LIN {X 0,Y 468.722,Z 59.104,A -85,B 0,C 180,E1 -7454.434,E2 -7454.434} C_VEL
LIN {X 0,Y 467.684,Z 59.23,A -85,B 0,C 180,E1 -7455.151,E2 -7455.151} C_VEL
LIN {X 0,Y 467.596,Z 59.24,A -85,B 0,C 180,E1 -7455.394,E2 -7455.394} C_VEL
LIN {X 0,Y 467.647,Z 59.28,A -85,B 0,C 180,E1 -7456.807,E2 -7456.807} C_VEL
LIN {X 0,Y 468.564,Z 66.05,A -85,B 0,C 180,E1 -7458.318,E2 -7458.318} C_VEL
LIN {X 0,Y 468.563,Z 74.796,A -85,B 0,C 180,E1 -7460.187,E2 -7460.187} C_VEL
LIN {X 0,Y 471.18,Z 89.776,A -85,B 0,C 180,E1 -7460.508,E2 -7460.508} C_VEL
LIN {X 0,Y 470.424,Z 181.464,A -85,B 0,C 180,E1 -7461.922,E2 -7461.922} C_VEL
LIN {X 0,Y 470.218,Z 194.57,A -85,B 0,C 180,E1 -7462.297,E2 -7462.297} C_VEL
LIN {X 0,Y 469.826,Z 207.741,A -85,B 0,C 180,E1 -7462.857,E2 -7462.857} C_VEL
LIN {X 0,Y 469.579,Z 219.557,A -85,B 0,C 180,E1 -7463.555,E2 -7463.555} C_VEL
LIN {X 0,Y 469.031,Z 230.914,A -85,B 0,C 180,E1 -7464.411,E2 -7464.411} C_VEL
LIN {X 0,Y 468.581,Z 241.141,A -85,B 0,C 180,E1 -7465.376,E2 -7465.376} C_VEL
LIN {X 0,Y 468.212,Z 249.513,A -85,B 0,C 180,E1 -7466.343,E2 -7466.343} C_VEL
LIN {X 0,Y 467.732,Z 258.606,A -85,B 0,C 180,E1 -7467.632,E2 -7467.632} C_VEL
LIN {X 0,Y 467.395,Z 265.922,A -85,B 0,C 180,E1 -7468.923,E2 -7468.923} C_VEL
LIN {X 0,Y 467.046,Z 272.679,A -85,B 0,C 180,E1 -7470.431,E2 -7470.431} C_VEL
LIN {X 0,Y 466.837,Z 277.14,A -85,B 0,C 180,E1 -7471.726,E2 -7471.726} C_VEL
LIN {X 0,Y 466.857,Z 279.486,A -85,B 0,C 180,E1 -7472.589,E2 -7472.589} C_VEL
LIN {X 0,Y 466.812,Z 281.417,A -85,B 0,C 180,E1 -7473.453,E2 -7473.453} C_VEL
LIN {X 0,Y 466.694,Z 282.945,A -85,B 0,C 180,E1 -7474.318,E2 -7474.318} C_VEL
LIN {X 0,Y 466.717,Z 284.018,A -85,B 0,C 180,E1 -7475.184,E2 -7475.184} C_VEL
LIN {X 0,Y 466.747,Z 284.88,A -85,B 0,C 180,E1 -7476.385,E2 -7476.385} C_VEL
LIN {X 0,Y 466.689,Z 284.914,A -85,B 0,C 180,E1 -7477.79,E2 -7477.79} C_VEL
LIN {X 0,Y 466.685,Z 284.397,A -85,B 0,C 180,E1 -7478.662,E2 -7478.662} C_VEL
LIN {X 0,Y 466.724,Z 282.165,A -85,B 0,C 180,E1 -7480.411,E2 -7480.411} C_VEL
LIN {X 0,Y 466.916,Z 278.848,A -85,B 0,C 180,E1 -7481.934,E2 -7481.934} C_VEL
LIN {X 0,Y 467.093,Z 273.978,A -85,B 0,C 180,E1 -7483.487,E2 -7483.487} C_VEL
LIN {X 0,Y 467.477,Z 267.522,A -85,B 0,C 180,E1 -7485.031,E2 -7485.031} C_VEL
LIN {X 0,Y 467.808,Z 260.476,A -85,B 0,C 180,E1 -7486.349,E2 -7486.349} C_VEL
LIN {X 0,Y 468.253,Z 251.445,A -85,B 0,C 180,E1 -7487.694,E2 -7487.694} C_VEL
LIN {X 0,Y 468.777,Z 242.455,A -85,B 0,C 180,E1 -7488.777,E2 -7488.777} C_VEL
LIN {X 0,Y 469.253,Z 231.889,A -85,B 0,C 180,E1 -7489.807,E2 -7489.807} C_VEL
LIN {X 0,Y 469.773,Z 220.35,A -85,B 0,C 180,E1 -7490.698,E2 -7490.698} C_VEL
LIN {X 0,Y 470.294,Z 208.288,A -85,B 0,C 180,E1 -7491.42,E2 -7491.42} C_VEL
LIN {X 0,Y 470.684,Z 195.785,A -85,B 0,C 180,E1 -7491.967,E2 -7491.967} C_VEL
LIN {X 0,Y 470.974,Z 182.953,A -85,B 0,C 180,E1 -7492.349,E2 -7492.349} C_VEL
LIN {X 0,Y 471.195,Z 149.03,A -85,B 0,C 180,E1 -7492.905,E2 -7492.905} C_VEL
LIN {X 0,Y 471.683,Z 88.302,A -85,B 0,C 180,E1 -7493.841,E2 -7493.841} C_VEL
LIN {X 0,Y 468.749,Z 74.914,A -85,B 0,C 180,E1 -7494.191,E2 -7494.191} C_VEL
LIN {X 0,Y 468.9,Z 66.893,A -85,B 0,C 180,E1 -7495.933,E2 -7495.933} C_VEL
LIN {X 0,Y 467.611,Z 59.24,A -85,B 0,C 180,E1 -7497.729,E2 -7497.729} C_VEL
LIN {X 0,Y 467.544,Z 59.245,A -85,B 0,C 180,E1 -7501.039,E2 -7501.039} C_VEL
LIN {X 0,Y 467.566,Z 59.245,A -85,B 0,C 180,E1 -7504.237,E2 -7504.237} C_VEL
LIN {X 0,Y 467.516,Z 59.246,A -85,B 0,C 180,E1 -7507.18,E2 -7507.18} C_VEL
LIN {X 0,Y 467.541,Z 59.247,A -85,B 0,C 180,E1 -7510.269,E2 -7510.269} C_VEL
LIN {X 0,Y 467.519,Z 59.247,A -85,B 0,C 180,E1 -7512.568,E2 -7512.568} C_VEL
LIN {X 0,Y 467.565,Z 59.232,A -85,B 0,C 180,E1 -7515.052,E2 -7515.052} C_VEL
LIN {X 0,Y 467.553,Z 59.239,A -85,B 0,C 180,E1 -7518.727,E2 -7518.727} C_VEL
LIN {X 0,Y 467.534,Z 59.246,A -85,B 0,C 180,E1 -7521.952,E2 -7521.952} C_VEL
LIN {X 0,Y 467.543,Z 59.244,A -85,B 0,C 180,E1 -7525.165,E2 -7525.165} C_VEL
LIN {X 0,Y 467.545,Z 59.239,A -85,B 0,C 180,E1 -7528.257,E2 -7528.257} C_VEL
LIN {X 0,Y 467.53,Z 59.248,A -85,B 0,C 180,E1 -7531.247,E2 -7531.247} C_VEL
LIN {X 0,Y 467.564,Z 59.24,A -85,B 0,C 180,E1 -7534.405,E2 -7534.405} C_VEL
LIN {X 0,Y 467.575,Z 59.24,A -85,B 0,C 180,E1 -7536.995,E2 -7536.995} C_VEL
LIN {X 0,Y 467.623,Z 59.232,A -85,B 0,C 180,E1 -7539.777,E2 -7539.777} C_VEL
LIN {X 0,Y 467.594,Z 59.236,A -85,B 0,C 180,E1 -7542.506,E2 -7542.506} C_VEL
LIN {X 0,Y 467.598,Z 59.237,A -85,B 0,C 180,E1 -7545.196,E2 -7545.196} C_VEL
LIN {X 0,Y 467.659,Z 59.223,A -85,B 0,C 180,E1 -7547.854,E2 -7547.854} C_VEL
LIN {X 0,Y 467.66,Z 59.228,A -85,B 0,C 180,E1 -7551.357,E2 -7551.357} C_VEL
LIN {X 0,Y 467.696,Z 59.22,A -85,B 0,C 180,E1 -7553.962,E2 -7553.962} C_VEL
LIN {X 0,Y 467.826,Z 59.207,A -85,B 0,C 180,E1 -7557.417,E2 -7557.417} C_VEL
LIN {X 0,Y 467.852,Z 59.203,A -85,B 0,C 180,E1 -7560,E2 -7560} C_VEL
LIN {X 0,Y 467.816,Z 59.21,A -85,B 0,C 180,E1 -7562.583,E2 -7562.583} C_VEL
LIN {X 0,Y 467.706,Z 59.221,A -85,B 0,C 180,E1 -7566.038,E2 -7566.038} C_VEL
LIN {X 0,Y 467.661,Z 59.227,A -85,B 0,C 180,E1 -7568.643,E2 -7568.643} C_VEL
LIN {X 0,Y 467.66,Z 59.227,A -85,B 0,C 180,E1 -7572.145,E2 -7572.145} C_VEL
LIN {X 0,Y 467.64,Z 59.233,A -85,B 0,C 180,E1 -7575.695,E2 -7575.695} C_VEL
LIN {X 0,Y 467.623,Z 59.236,A -85,B 0,C 180,E1 -7579.308,E2 -7579.308} C_VEL
LIN {X 0,Y 467.537,Z 59.239,A -85,B 0,C 180,E1 -7582.074,E2 -7582.074} C_VEL
LIN {X 0,Y 467.572,Z 59.242,A -85,B 0,C 180,E1 -7584.889,E2 -7584.889} C_VEL
LIN {X 0,Y 467.618,Z 59.234,A -85,B 0,C 180,E1 -7587.769,E2 -7587.769} C_VEL
LIN {X 0,Y 467.57,Z 59.242,A -85,B 0,C 180,E1 -7591.044,E2 -7591.044} C_VEL
LIN {X 0,Y 467.591,Z 59.236,A -85,B 0,C 180,E1 -7594.242,E2 -7594.242} C_VEL
LIN {X 0,Y 467.55,Z 59.238,A -85,B 0,C 180,E1 -7597.186,E2 -7597.186} C_VEL
LIN {X 0,Y 467.577,Z 59.241,A -85,B 0,C 180,E1 -7600.265,E2 -7600.265} C_VEL
LIN {X 0,Y 467.589,Z 59.243,A -85,B 0,C 180,E1 -7602.567,E2 -7602.567} C_VEL
LIN {X 0,Y 467.568,Z 59.241,A -85,B 0,C 180,E1 -7605.052,E2 -7605.052} C_VEL
LIN {X 0,Y 467.592,Z 59.235,A -85,B 0,C 180,E1 -7607.44,E2 -7607.44} C_VEL
LIN {X 0,Y 467.585,Z 59.239,A -85,B 0,C 180,E1 -7610.855,E2 -7610.855} C_VEL
LIN {X 0,Y 467.562,Z 59.242,A -85,B 0,C 180,E1 -7614.261,E2 -7614.261} C_VEL
LIN {X 0,Y 467.585,Z 59.242,A -85,B 0,C 180,E1 -7617.321,E2 -7617.321} C_VEL
LIN {X 0,Y 467.572,Z 59.244,A -85,B 0,C 180,E1 -7620.667,E2 -7620.667} C_VEL
LIN {X 0,Y 467.696,Z 59.391,A -85,B 0,C 180,E1 -7623.295,E2 -7623.295} C_VEL
LIN {X 0,Y 470.046,Z 71.407,A -85,B 0,C 180,E1 -7625.579,E2 -7625.579} C_VEL
LIN {X 0,Y 469.737,Z 81.506,A -85,B 0,C 180,E1 -7627.34,E2 -7627.34} C_VEL
LIN {X 0,Y 468.798,Z 101.855,A -85,B 0,C 180,E1 -7630.816,E2 -7630.816} C_VEL
LIN {X 0,Y 468.334,Z 113.848,A -85,B 0,C 180,E1 -7632.842,E2 -7632.842} C_VEL
LIN {X 0,Y 471.406,Z 134.719,A -85,B 0,C 180,E1 -7633.296,E2 -7633.296} C_VEL
LIN {X 0,Y 470.758,Z 222.171,A -85,B 0,C 180,E1 -7634.661,E2 -7634.661} C_VEL
LIN {X 0,Y 470.321,Z 235.512,A -85,B 0,C 180,E1 -7635.034,E2 -7635.034} C_VEL
LIN {X 0,Y 469.848,Z 247.706,A -85,B 0,C 180,E1 -7635.545,E2 -7635.545} C_VEL
LIN {X 0,Y 469.32,Z 260.024,A -85,B 0,C 180,E1 -7636.247,E2 -7636.247} C_VEL
LIN {X 0,Y 468.688,Z 271.899,A -85,B 0,C 180,E1 -7637.133,E2 -7637.133} C_VEL
LIN {X 0,Y 468.246,Z 282.11,A -85,B 0,C 180,E1 -7638.09,E2 -7638.09} C_VEL
LIN {X 0,Y 467.715,Z 291.557,A -85,B 0,C 180,E1 -7639.174,E2 -7639.174} C_VEL
LIN {X 0,Y 467.305,Z 300.678,A -85,B 0,C 180,E1 -7640.477,E2 -7640.477} C_VEL
LIN {X 0,Y 466.988,Z 308.043,A -85,B 0,C 180,E1 -7641.78,E2 -7641.78} C_VEL
LIN {X 0,Y 466.824,Z 313.963,A -85,B 0,C 180,E1 -7643.082,E2 -7643.082} C_VEL
LIN {X 0,Y 466.709,Z 318.64,A -85,B 0,C 180,E1 -7644.383,E2 -7644.383} C_VEL
LIN {X 0,Y 466.646,Z 322.21,A -85,B 0,C 180,E1 -7645.681,E2 -7645.681} C_VEL
LIN {X 0,Y 466.699,Z 324.041,A -85,B 0,C 180,E1 -7646.546,E2 -7646.546} C_VEL
LIN {X 0,Y 466.684,Z 325.418,A -85,B 0,C 180,E1 -7647.41,E2 -7647.41} C_VEL
LIN {X 0,Y 466.664,Z 326.4,A -85,B 0,C 180,E1 -7648.274,E2 -7648.274} C_VEL
LIN {X 0,Y 466.63,Z 326.992,A -85,B 0,C 180,E1 -7649.137,E2 -7649.137} C_VEL
LIN {X 0,Y 466.614,Z 327.175,A -85,B 0,C 180,E1 -7650,E2 -7650} C_VEL
LIN {X 0,Y 466.664,Z 326.308,A -85,B 0,C 180,E1 -7651.726,E2 -7651.726} C_VEL
LIN {X 0,Y 466.685,Z 325.29,A -85,B 0,C 180,E1 -7652.589,E2 -7652.589} C_VEL
LIN {X 0,Y 466.73,Z 323.852,A -85,B 0,C 180,E1 -7653.453,E2 -7653.453} C_VEL
LIN {X 0,Y 466.685,Z 320.859,A -85,B 0,C 180,E1 -7654.751,E2 -7654.751} C_VEL
LIN {X 0,Y 466.704,Z 315.725,A -85,B 0,C 180,E1 -7656.341,E2 -7656.341} C_VEL
LIN {X 0,Y 466.927,Z 309.562,A -85,B 0,C 180,E1 -7657.785,E2 -7657.785} C_VEL
LIN {X 0,Y 467.158,Z 302.53,A -85,B 0,C 180,E1 -7659.088,E2 -7659.088} C_VEL
LIN {X 0,Y 467.465,Z 293.71,A -85,B 0,C 180,E1 -7660.393,E2 -7660.393} C_VEL
LIN {X 0,Y 468.005,Z 283.701,A -85,B 0,C 180,E1 -7661.587,E2 -7661.587} C_VEL
LIN {X 0,Y 468.432,Z 273.768,A -85,B 0,C 180,E1 -7662.542,E2 -7662.542} C_VEL
LIN {X 0,Y 468.936,Z 262.165,A -85,B 0,C 180,E1 -7663.432,E2 -7663.432} C_VEL
LIN {X 0,Y 469.429,Z 250.422,A -85,B 0,C 180,E1 -7664.136,E2 -7664.136} C_VEL
LIN {X 0,Y 469.88,Z 237.655,A -85,B 0,C 180,E1 -7664.702,E2 -7664.702} C_VEL
LIN {X 0,Y 470.294,Z 224.05,A -85,B 0,C 180,E1 -7665.104,E2 -7665.104} C_VEL
LIN {X 0,Y 470.602,Z 188.382,A -85,B 0,C 180,E1 -7665.677,E2 -7665.677} C_VEL
LIN {X 0,Y 470.79,Z 132.877,A -85,B 0,C 180,E1 -7666.528,E2 -7666.528} C_VEL
LIN {X 0,Y 468.138,Z 113.96,A -85,B 0,C 180,E1 -7666.918,E2 -7666.918} C_VEL
LIN {X 0,Y 468.755,Z 95.783,A -85,B 0,C 180,E1 -7669.943,E2 -7669.943} C_VEL
LIN {X 0,Y 469.614,Z 75.42,A -85,B 0,C 180,E1 -7673.365,E2 -7673.365} C_VEL
LIN {X 0,Y 469.599,Z 69.43,A -85,B 0,C 180,E1 -7674.394,E2 -7674.394} C_VEL
LIN {X 0,Y 467.643,Z 59.237,A -85,B 0,C 180,E1 -7676.257,E2 -7676.257} C_VEL
LIN {X 0,Y 467.571,Z 59.242,A -85,B 0,C 180,E1 -7679.332,E2 -7679.332} C_VEL
LIN {X 0,Y 467.582,Z 59.237,A -85,B 0,C 180,E1 -7682.679,E2 -7682.679} C_VEL
LIN {X 0,Y 467.56,Z 59.247,A -85,B 0,C 180,E1 -7685.739,E2 -7685.739} C_VEL
LIN {X 0,Y 467.583,Z 59.238,A -85,B 0,C 180,E1 -7689.144,E2 -7689.144} C_VEL
LIN {X 0,Y 467.586,Z 59.236,A -85,B 0,C 180,E1 -7692.567,E2 -7692.567} C_VEL
LIN {X 0,Y 467.565,Z 59.241,A -85,B 0,C 180,E1 -7695.052,E2 -7695.052} C_VEL
LIN {X 0,Y 467.588,Z 59.244,A -85,B 0,C 180,E1 -7697.44,E2 -7697.44} C_VEL
LIN {X 0,Y 467.575,Z 59.24,A -85,B 0,C 180,E1 -7700.855,E2 -7700.855} C_VEL
LIN {X 0,Y 467.56,Z 59.239,A -85,B 0,C 180,E1 -7704.261,E2 -7704.261} C_VEL
LIN {X 0,Y 467.581,Z 59.242,A -85,B 0,C 180,E1 -7707.321,E2 -7707.321} C_VEL
LIN {X 0,Y 467.569,Z 59.242,A -85,B 0,C 180,E1 -7710.667,E2 -7710.667} C_VEL
LIN {X 0,Y 467.616,Z 59.237,A -85,B 0,C 180,E1 -7713.2,E2 -7713.2} C_VEL
LIN {X 0,Y 467.591,Z 59.239,A -85,B 0,C 180,E1 -7716.468,E2 -7716.468} C_VEL
LIN {X 0,Y 467.622,Z 59.232,A -85,B 0,C 180,E1 -7719.777,E2 -7719.777} C_VEL
LIN {X 0,Y 467.597,Z 59.241,A -85,B 0,C 180,E1 -7722.506,E2 -7722.506} C_VEL
LIN {X 0,Y 467.604,Z 59.235,A -85,B 0,C 180,E1 -7725.196,E2 -7725.196} C_VEL
LIN {X 0,Y 467.656,Z 59.229,A -85,B 0,C 180,E1 -7727.855,E2 -7727.855} C_VEL
LIN {X 0,Y 467.679,Z 59.224,A -85,B 0,C 180,E1 -7731.357,E2 -7731.357} C_VEL
LIN {X 0,Y 467.736,Z 59.221,A -85,B 0,C 180,E1 -7733.963,E2 -7733.963} C_VEL
LIN {X 0,Y 467.852,Z 59.203,A -85,B 0,C 180,E1 -7737.417,E2 -7737.417} C_VEL
LIN {X 0,Y 467.881,Z 59.206,A -85,B 0,C 180,E1 -7740,E2 -7740} C_VEL
LIN {X 0,Y 467.852,Z 59.204,A -85,B 0,C 180,E1 -7742.583,E2 -7742.583} C_VEL
LIN {X 0,Y 467.721,Z 59.225,A -85,B 0,C 180,E1 -7746.038,E2 -7746.038} C_VEL
LIN {X 0,Y 467.669,Z 59.226,A -85,B 0,C 180,E1 -7748.643,E2 -7748.643} C_VEL
LIN {X 0,Y 467.656,Z 59.23,A -85,B 0,C 180,E1 -7752.146,E2 -7752.146} C_VEL
LIN {X 0,Y 467.639,Z 59.236,A -85,B 0,C 180,E1 -7755.695,E2 -7755.695} C_VEL
LIN {X 0,Y 467.621,Z 59.237,A -85,B 0,C 180,E1 -7759.308,E2 -7759.308} C_VEL
LIN {X 0,Y 467.534,Z 59.243,A -85,B 0,C 180,E1 -7762.074,E2 -7762.074} C_VEL
LIN {X 0,Y 467.569,Z 59.241,A -85,B 0,C 180,E1 -7764.89,E2 -7764.89} C_VEL
LIN {X 0,Y 467.616,Z 59.234,A -85,B 0,C 180,E1 -7767.77,E2 -7767.77} C_VEL
LIN {X 0,Y 467.568,Z 59.246,A -85,B 0,C 180,E1 -7771.045,E2 -7771.045} C_VEL
LIN {X 0,Y 467.578,Z 59.237,A -85,B 0,C 180,E1 -7774.241,E2 -7774.241} C_VEL
LIN {X 0,Y 467.548,Z 59.245,A -85,B 0,C 180,E1 -7777.187,E2 -7777.187} C_VEL
LIN {X 0,Y 467.559,Z 59.241,A -85,B 0,C 180,E1 -7780.267,E2 -7780.267} C_VEL
LIN {X 0,Y 467.547,Z 59.241,A -85,B 0,C 180,E1 -7783.746,E2 -7783.746} C_VEL
LIN {X 0,Y 467.55,Z 59.244,A -85,B 0,C 180,E1 -7786.255,E2 -7786.255} C_VEL
LIN {X 0,Y 467.572,Z 59.238,A -85,B 0,C 180,E1 -7789.735,E2 -7789.735} C_VEL
LIN {X 0,Y 467.543,Z 59.244,A -85,B 0,C 180,E1 -7792.815,E2 -7792.815} C_VEL
LIN {X 0,Y 467.586,Z 59.243,A -85,B 0,C 180,E1 -7796.212,E2 -7796.212} C_VEL
LIN {X 0,Y 467.572,Z 59.238,A -85,B 0,C 180,E1 -7799.267,E2 -7799.267} C_VEL
LIN {X 0,Y 467.606,Z 59.237,A -85,B 0,C 180,E1 -7802.469,E2 -7802.469} C_VEL
LIN {X 0,Y 467.563,Z 59.239,A -85,B 0,C 180,E1 -7805.111,E2 -7805.111} C_VEL
LIN {X 0,Y 467.538,Z 59.25,A -85,B 0,C 180,E1 -7807.927,E2 -7807.927} C_VEL
LIN {X 0,Y 467.624,Z 59.232,A -85,B 0,C 180,E1 -7810.693,E2 -7810.693} C_VEL
LIN {X 0,Y 467.642,Z 59.235,A -85,B 0,C 180,E1 -7814.305,E2 -7814.305} C_VEL
LIN {X 0,Y 467.596,Z 59.24,A -85,B 0,C 180,E1 -7815.394,E2 -7815.394} C_VEL
LIN {X 0,Y 466.953,Z 59.509,A -85,B 0,C 180,E1 -7815.879,E2 -7815.879} C_VEL
LIN {X 0,Y 465.485,Z 60.23,A -85,B 0,C 180,E1 -7816.337,E2 -7816.337} C_VEL
LIN {X 0,Y 462.208,Z 62.778,A -85,B 0,C 180,E1 -7817.211,E2 -7817.211} C_VEL
LIN {X 0,Y 461.41,Z 64.535,A -85,B 0,C 180,E1 -7817.652,E2 -7817.652} C_VEL
LIN {X 0,Y 461.411,Z 65.177,A -85,B 0,C 180,E1 -7817.799,E2 -7817.799} C_VEL
LIN {X 0,Y 461.656,Z 70.789,A -85,B 0,C 180,E1 -7819.03,E2 -7819.03} C_VEL
LIN {X 0,Y 461.573,Z 75.069,A -85,B 0,C 180,E1 -7819.949,E2 -7819.949} C_VEL
LIN {X 0,Y 464.328,Z 89.869,A -85,B 0,C 180,E1 -7820.28,E2 -7820.28} C_VEL
LIN {X 0,Y 463.544,Z 181.792,A -85,B 0,C 180,E1 -7821.719,E2 -7821.719} C_VEL
LIN {X 0,Y 463.316,Z 194.898,A -85,B 0,C 180,E1 -7822.099,E2 -7822.099} C_VEL
LIN {X 0,Y 462.945,Z 207.508,A -85,B 0,C 180,E1 -7822.641,E2 -7822.641} C_VEL
LIN {X 0,Y 462.674,Z 219.492,A -85,B 0,C 180,E1 -7823.349,E2 -7823.349} C_VEL
LIN {X 0,Y 462.089,Z 230.925,A -85,B 0,C 180,E1 -7824.217,E2 -7824.217} C_VEL
LIN {X 0,Y 461.612,Z 241.208,A -85,B 0,C 180,E1 -7825.197,E2 -7825.197} C_VEL
LIN {X 0,Y 461.172,Z 250.479,A -85,B 0,C 180,E1 -7826.287,E2 -7826.287} C_VEL
LIN {X 0,Y 460.677,Z 259.439,A -85,B 0,C 180,E1 -7827.596,E2 -7827.596} C_VEL
LIN {X 0,Y 460.337,Z 266.666,A -85,B 0,C 180,E1 -7828.907,E2 -7828.907} C_VEL
LIN {X 0,Y 460.037,Z 271.577,A -85,B 0,C 180,E1 -7830,E2 -7830} C_VEL
LIN {X 0,Y 459.82,Z 276.346,A -85,B 0,C 180,E1 -7831.314,E2 -7831.314} C_VEL
LIN {X 0,Y 459.765,Z 280.011,A -85,B 0,C 180,E1 -7832.629,E2 -7832.629} C_VEL
LIN {X 0,Y 459.735,Z 281.909,A -85,B 0,C 180,E1 -7833.506,E2 -7833.506} C_VEL
LIN {X 0,Y 459.603,Z 283.385,A -85,B 0,C 180,E1 -7834.385,E2 -7834.385} C_VEL
LIN {X 0,Y 459.65,Z 284.414,A -85,B 0,C 180,E1 -7835.264,E2 -7835.264} C_VEL
LIN {X 0,Y 459.676,Z 285.194,A -85,B 0,C 180,E1 -7836.385,E2 -7836.385} C_VEL
LIN {X 0,Y 459.607,Z 285.2,A -85,B 0,C 180,E1 -7837.911,E2 -7837.911} C_VEL
LIN {X 0,Y 459.577,Z 283.693,A -85,B 0,C 180,E1 -7839.684,E2 -7839.684} C_VEL
LIN {X 0,Y 459.665,Z 282.346,A -85,B 0,C 180,E1 -7840.572,E2 -7840.572} C_VEL
LIN {X 0,Y 459.849,Z 279.251,A -85,B 0,C 180,E1 -7842.002,E2 -7842.002} C_VEL
LIN {X 0,Y 460.014,Z 275.565,A -85,B 0,C 180,E1 -7843.248,E2 -7843.248} C_VEL
LIN {X 0,Y 460.379,Z 269.486,A -85,B 0,C 180,E1 -7844.815,E2 -7844.815} C_VEL
LIN {X 0,Y 460.682,Z 263.523,A -85,B 0,C 180,E1 -7846.031,E2 -7846.031} C_VEL
LIN {X 0,Y 461.074,Z 255.92,A -85,B 0,C 180,E1 -7847.292,E2 -7847.292} C_VEL
LIN {X 0,Y 461.57,Z 247.605,A -85,B 0,C 180,E1 -7848.418,E2 -7848.418} C_VEL
LIN {X 0,Y 462.105,Z 237.37,A -85,B 0,C 180,E1 -7849.548,E2 -7849.548} C_VEL
LIN {X 0,Y 462.623,Z 227.142,A -85,B 0,C 180,E1 -7850.451,E2 -7850.451} C_VEL
LIN {X 0,Y 463.184,Z 215.944,A -85,B 0,C 180,E1 -7851.239,E2 -7851.239} C_VEL
LIN {X 0,Y 463.675,Z 203.439,A -85,B 0,C 180,E1 -7851.916,E2 -7851.916} C_VEL
LIN {X 0,Y 464.037,Z 190.348,A -85,B 0,C 180,E1 -7852.414,E2 -7852.414} C_VEL
LIN {X 0,Y 464.262,Z 177.871,A -85,B 0,C 180,E1 -7852.716,E2 -7852.716} C_VEL
LIN {X 0,Y 464.945,Z 89.046,A -85,B 0,C 180,E1 -7854.114,E2 -7854.114} C_VEL
LIN {X 0,Y 461.826,Z 75.168,A -85,B 0,C 180,E1 -7854.498,E2 -7854.498} C_VEL
LIN {X 0,Y 461.88,Z 67.524,A -85,B 0,C 180,E1 -7856.185,E2 -7856.185} C_VEL
LIN {X 0,Y 460.562,Z 60.117,A -85,B 0,C 180,E1 -7857.944,E2 -7857.944} C_VEL
LIN {X 0,Y 460.499,Z 60.122,A -85,B 0,C 180,E1 -7861.277,E2 -7861.277} C_VEL
LIN {X 0,Y 460.511,Z 60.121,A -85,B 0,C 180,E1 -7864.501,E2 -7864.501} C_VEL
LIN {X 0,Y 460.484,Z 60.123,A -85,B 0,C 180,E1 -7867.625,E2 -7867.625} C_VEL
LIN {X 0,Y 460.507,Z 60.12,A -85,B 0,C 180,E1 -7871.014,E2 -7871.014} C_VEL
LIN {X 0,Y 460.509,Z 60.111,A -85,B 0,C 180,E1 -7874.59,E2 -7874.59} C_VEL
LIN {X 0,Y 460.474,Z 60.127,A -85,B 0,C 180,E1 -7877.812,E2 -7877.812} C_VEL
LIN {X 0,Y 460.476,Z 60.124,A -85,B 0,C 180,E1 -7880.131,E2 -7880.131} C_VEL
LIN {X 0,Y 460.456,Z 60.131,A -85,B 0,C 180,E1 -7883.468,E2 -7883.468} C_VEL
LIN {X 0,Y 460.503,Z 60.12,A -85,B 0,C 180,E1 -7886.673,E2 -7886.673} C_VEL
LIN {X 0,Y 460.482,Z 60.124,A -85,B 0,C 180,E1 -7889.757,E2 -7889.757} C_VEL
LIN {X 0,Y 460.487,Z 60.121,A -85,B 0,C 180,E1 -7892.75,E2 -7892.75} C_VEL
LIN {X 0,Y 460.515,Z 60.118,A -85,B 0,C 180,E1 -7895.666,E2 -7895.666} C_VEL
LIN {X 0,Y 460.525,Z 60.116,A -85,B 0,C 180,E1 -7898.578,E2 -7898.578} C_VEL
LIN {X 0,Y 460.587,Z 60.107,A -85,B 0,C 180,E1 -7901.31,E2 -7901.31} C_VEL
LIN {X 0,Y 460.589,Z 60.107,A -85,B 0,C 180,E1 -7904.058,E2 -7904.058} C_VEL
LIN {X 0,Y 460.613,Z 60.1,A -85,B 0,C 180,E1 -7907.666,E2 -7907.666} C_VEL
LIN {X 0,Y 460.612,Z 60.106,A -85,B 0,C 180,E1 -7911.223,E2 -7911.223} C_VEL
LIN {X 0,Y 460.663,Z 60.095,A -85,B 0,C 180,E1 -7913.869,E2 -7913.869} C_VEL
LIN {X 0,Y 460.77,Z 60.086,A -85,B 0,C 180,E1 -7917.377,E2 -7917.377} C_VEL
LIN {X 0,Y 460.822,Z 60.078,A -85,B 0,C 180,E1 -7920,E2 -7920} C_VEL
LIN {X 0,Y 460.76,Z 60.089,A -85,B 0,C 180,E1 -7922.623,E2 -7922.623} C_VEL
LIN {X 0,Y 460.672,Z 60.097,A -85,B 0,C 180,E1 -7926.13,E2 -7926.13} C_VEL
LIN {X 0,Y 460.613,Z 60.105,A -85,B 0,C 180,E1 -7928.776,E2 -7928.776} C_VEL
LIN {X 0,Y 460.613,Z 60.103,A -85,B 0,C 180,E1 -7932.334,E2 -7932.334} C_VEL
LIN {X 0,Y 460.582,Z 60.108,A -85,B 0,C 180,E1 -7935.988,E2 -7935.988} C_VEL
LIN {X 0,Y 460.569,Z 60.116,A -85,B 0,C 180,E1 -7939.615,E2 -7939.615} C_VEL
LIN {X 0,Y 460.513,Z 60.113,A -85,B 0,C 180,E1 -7942.428,E2 -7942.428} C_VEL
LIN {X 0,Y 460.548,Z 60.113,A -85,B 0,C 180,E1 -7945.796,E2 -7945.796} C_VEL
LIN {X 0,Y 460.552,Z 60.113,A -85,B 0,C 180,E1 -7948.233,E2 -7948.233} C_VEL
LIN {X 0,Y 460.523,Z 60.12,A -85,B 0,C 180,E1 -7951.283,E2 -7951.283} C_VEL
LIN {X 0,Y 460.535,Z 60.117,A -85,B 0,C 180,E1 -7954.505,E2 -7954.505} C_VEL
LIN {X 0,Y 460.503,Z 60.115,A -85,B 0,C 180,E1 -7957.623,E2 -7957.623} C_VEL
LIN {X 0,Y 460.541,Z 60.117,A -85,B 0,C 180,E1 -7960.269,E2 -7960.269} C_VEL
LIN {X 0,Y 460.501,Z 60.12,A -85,B 0,C 180,E1 -7963.375,E2 -7963.375} C_VEL
LIN {X 0,Y 460.502,Z 60.124,A -85,B 0,C 180,E1 -7966.624,E2 -7966.624} C_VEL
LIN {X 0,Y 460.545,Z 60.114,A -85,B 0,C 180,E1 -7969.73,E2 -7969.73} C_VEL
LIN {X 0,Y 460.502,Z 60.125,A -85,B 0,C 180,E1 -7972.524,E2 -7972.524} C_VEL
LIN {X 0,Y 460.549,Z 60.116,A -85,B 0,C 180,E1 -7975.624,E2 -7975.624} C_VEL
LIN {X 0,Y 460.54,Z 60.121,A -85,B 0,C 180,E1 -7978.744,E2 -7978.744} C_VEL
LIN {X 0,Y 460.584,Z 60.116,A -85,B 0,C 180,E1 -7982.254,E2 -7982.254} C_VEL
LIN {X 0,Y 460.637,Z 60.118,A -85,B 0,C 180,E1 -7983.006,E2 -7983.006} C_VEL
LIN {X 0,Y 463.017,Z 72.017,A -85,B 0,C 180,E1 -7985.314,E2 -7985.314} C_VEL
LIN {X 0,Y 463.181,Z 76.078,A -85,B 0,C 180,E1 -7986.053,E2 -7986.053} C_VEL
LIN {X 0,Y 462.19,Z 94.646,A -85,B 0,C 180,E1 -7989.296,E2 -7989.296} C_VEL
LIN {X 0,Y 461.38,Z 113.462,A -85,B 0,C 180,E1 -7992.535,E2 -7992.535} C_VEL
LIN {X 0,Y 464.644,Z 135.081,A -85,B 0,C 180,E1 -7993.029,E2 -7993.029} C_VEL
LIN {X 0,Y 463.932,Z 222.939,A -85,B 0,C 180,E1 -7994.43,E2 -7994.43} C_VEL
LIN {X 0,Y 463.456,Z 236.668,A -85,B 0,C 180,E1 -7994.836,E2 -7994.836} C_VEL
LIN {X 0,Y 462.946,Z 249.012,A -85,B 0,C 180,E1 -7995.381,E2 -7995.381} C_VEL
LIN {X 0,Y 462.333,Z 261.647,A -85,B 0,C 180,E1 -7996.148,E2 -7996.148} C_VEL
LIN {X 0,Y 461.722,Z 272.491,A -85,B 0,C 180,E1 -7996.99,E2 -7996.99} C_VEL
LIN {X 0,Y 461.226,Z 283.069,A -85,B 0,C 180,E1 -7998.017,E2 -7998.017} C_VEL
LIN {X 0,Y 460.61,Z 293.05,A -85,B 0,C 180,E1 -7999.227,E2 -7999.227} C_VEL
LIN {X 0,Y 460.186,Z 301.861,A -85,B 0,C 180,E1 -8000.55,E2 -8000.55} C_VEL
LIN {X 0,Y 459.902,Z 308.923,A -85,B 0,C 180,E1 -8001.874,E2 -8001.874} C_VEL
LIN {X 0,Y 459.671,Z 315.395,A -85,B 0,C 180,E1 -8003.416,E2 -8003.416} C_VEL
LIN {X 0,Y 459.631,Z 319.672,A -85,B 0,C 180,E1 -8004.736,E2 -8004.736} C_VEL
LIN {X 0,Y 459.563,Z 321.942,A -85,B 0,C 180,E1 -8005.614,E2 -8005.614} C_VEL
LIN {X 0,Y 459.595,Z 323.755,A -85,B 0,C 180,E1 -8006.493,E2 -8006.493} C_VEL
LIN {X 0,Y 459.605,Z 325.125,A -85,B 0,C 180,E1 -8007.37,E2 -8007.37} C_VEL
LIN {X 0,Y 459.562,Z 326.684,A -85,B 0,C 180,E1 -8009.123,E2 -8009.123} C_VEL
LIN {X 0,Y 459.545,Z 326.852,A -85,B 0,C 180,E1 -8010,E2 -8010} C_VEL
LIN {X 0,Y 459.562,Z 326.604,A -85,B 0,C 180,E1 -8010.876,E2 -8010.876} C_VEL
LIN {X 0,Y 459.607,Z 324.942,A -85,B 0,C 180,E1 -8012.629,E2 -8012.629} C_VEL
LIN {X 0,Y 459.625,Z 323.486,A -85,B 0,C 180,E1 -8013.506,E2 -8013.506} C_VEL
LIN {X 0,Y 459.615,Z 320.48,A -85,B 0,C 180,E1 -8014.824,E2 -8014.824} C_VEL
LIN {X 0,Y 459.613,Z 315.769,A -85,B 0,C 180,E1 -8016.318,E2 -8016.318} C_VEL
LIN {X 0,Y 459.84,Z 310.155,A -85,B 0,C 180,E1 -8017.685,E2 -8017.685} C_VEL
LIN {X 0,Y 460.042,Z 303.334,A -85,B 0,C 180,E1 -8019.009,E2 -8019.009} C_VEL
LIN {X 0,Y 460.375,Z 294.855,A -85,B 0,C 180,E1 -8020.333,E2 -8020.333} C_VEL
LIN {X 0,Y 460.864,Z 286.119,A -85,B 0,C 180,E1 -8021.434,E2 -8021.434} C_VEL
LIN {X 0,Y 461.305,Z 276.306,A -85,B 0,C 180,E1 -8022.449,E2 -8022.449} C_VEL
LIN {X 0,Y 461.831,Z 264.64,A -85,B 0,C 180,E1 -8023.419,E2 -8023.419} C_VEL
LIN {X 0,Y 462.382,Z 252.65,A -85,B 0,C 180,E1 -8024.187,E2 -8024.187} C_VEL
LIN {X 0,Y 462.884,Z 240.159,A -85,B 0,C 180,E1 -8024.789,E2 -8024.789} C_VEL
LIN {X 0,Y 463.293,Z 227.229,A -85,B 0,C 180,E1 -8025.226,E2 -8025.226} C_VEL
LIN {X 0,Y 463.486,Z 213.395,A -85,B 0,C 180,E1 -8025.501,E2 -8025.501} C_VEL
LIN {X 0,Y 463.915,Z 133.392,A -85,B 0,C 180,E1 -8026.741,E2 -8026.741} C_VEL
LIN {X 0,Y 461.151,Z 113.625,A -85,B 0,C 180,E1 -8027.158,E2 -8027.158} C_VEL
LIN {X 0,Y 461.755,Z 96.65,A -85,B 0,C 180,E1 -8030.026,E2 -8030.026} C_VEL
LIN {X 0,Y 462.599,Z 77.652,A -85,B 0,C 180,E1 -8033.266,E2 -8033.266} C_VEL
LIN {X 0,Y 462.653,Z 70.829,A -85,B 0,C 180,E1 -8034.452,E2 -8034.452} C_VEL
LIN {X 0,Y 460.588,Z 60.116,A -85,B 0,C 180,E1 -8036.446,E2 -8036.446} C_VEL
LIN {X 0,Y 460.532,Z 60.121,A -85,B 0,C 180,E1 -8039.558,E2 -8039.558} C_VEL
LIN {X 0,Y 460.532,Z 60.118,A -85,B 0,C 180,E1 -8042.284,E2 -8042.284} C_VEL
LIN {X 0,Y 460.511,Z 60.121,A -85,B 0,C 180,E1 -8045.445,E2 -8045.445} C_VEL
LIN {X 0,Y 460.545,Z 60.113,A -85,B 0,C 180,E1 -8048.898,E2 -8048.898} C_VEL
LIN {X 0,Y 460.523,Z 60.117,A -85,B 0,C 180,E1 -8052.181,E2 -8052.181} C_VEL
LIN {X 0,Y 460.513,Z 60.124,A -85,B 0,C 180,E1 -8055.411,E2 -8055.411} C_VEL
LIN {X 0,Y 460.531,Z 60.115,A -85,B 0,C 180,E1 -8058.397,E2 -8058.397} C_VEL
LIN {X 0,Y 460.523,Z 60.123,A -85,B 0,C 180,E1 -8061.267,E2 -8061.267} C_VEL
LIN {X 0,Y 460.511,Z 60.118,A -85,B 0,C 180,E1 -8064.554,E2 -8064.554} C_VEL
LIN {X 0,Y 460.531,Z 60.116,A -85,B 0,C 180,E1 -8067.716,E2 -8067.716} C_VEL
LIN {X 0,Y 460.539,Z 60.119,A -85,B 0,C 180,E1 -8070.769,E2 -8070.769} C_VEL
LIN {X 0,Y 460.562,Z 60.111,A -85,B 0,C 180,E1 -8073.735,E2 -8073.735} C_VEL
LIN {X 0,Y 460.545,Z 60.118,A -85,B 0,C 180,E1 -8076.624,E2 -8076.624} C_VEL
LIN {X 0,Y 460.55,Z 60.113,A -85,B 0,C 180,E1 -8079.453,E2 -8079.453} C_VEL
LIN {X 0,Y 460.549,Z 60.115,A -85,B 0,C 180,E1 -8082.23,E2 -8082.23} C_VEL
LIN {X 0,Y 460.564,Z 60.114,A -85,B 0,C 180,E1 -8084.965,E2 -8084.965} C_VEL
LIN {X 0,Y 460.609,Z 60.112,A -85,B 0,C 180,E1 -8088.559,E2 -8088.559} C_VEL
LIN {X 0,Y 460.695,Z 60.099,A -85,B 0,C 180,E1 -8092.109,E2 -8092.109} C_VEL
LIN {X 0,Y 460.694,Z 60.097,A -85,B 0,C 180,E1 -8094.748,E2 -8094.748} C_VEL
LIN {X 0,Y 460.792,Z 60.083,A -85,B 0,C 180,E1 -8097.378,E2 -8097.378} C_VEL
LIN {X 0,Y 460.851,Z 60.082,A -85,B 0,C 180,E1 -8100,E2 -8100} C_VEL
LIN {X 0,Y 460.792,Z 60.084,A -85,B 0,C 180,E1 -8102.623,E2 -8102.623} C_VEL
LIN {X 0,Y 460.685,Z 60.101,A -85,B 0,C 180,E1 -8106.13,E2 -8106.13} C_VEL
LIN {X 0,Y 460.619,Z 60.104,A -85,B 0,C 180,E1 -8108.777,E2 -8108.777} C_VEL
LIN {X 0,Y 460.614,Z 60.105,A -85,B 0,C 180,E1 -8112.445,E2 -8112.445} C_VEL
LIN {X 0,Y 460.601,Z 60.109,A -85,B 0,C 180,E1 -8115.998,E2 -8115.998} C_VEL
LIN {X 0,Y 460.567,Z 60.116,A -85,B 0,C 180,E1 -8119.616,E2 -8119.616} C_VEL
LIN {X 0,Y 460.51,Z 60.117,A -85,B 0,C 180,E1 -8122.429,E2 -8122.429} C_VEL
LIN {X 0,Y 460.546,Z 60.115,A -85,B 0,C 180,E1 -8125.797,E2 -8125.797} C_VEL
LIN {X 0,Y 460.55,Z 60.113,A -85,B 0,C 180,E1 -8128.234,E2 -8128.234} C_VEL
LIN {X 0,Y 460.521,Z 60.122,A -85,B 0,C 180,E1 -8131.283,E2 -8131.283} C_VEL
LIN {X 0,Y 460.524,Z 60.118,A -85,B 0,C 180,E1 -8134.504,E2 -8134.504} C_VEL
LIN {X 0,Y 460.501,Z 60.119,A -85,B 0,C 180,E1 -8137.624,E2 -8137.624} C_VEL
LIN {X 0,Y 460.525,Z 60.117,A -85,B 0,C 180,E1 -8140.267,E2 -8140.267} C_VEL
LIN {X 0,Y 460.504,Z 60.119,A -85,B 0,C 180,E1 -8143.376,E2 -8143.376} C_VEL
LIN {X 0,Y 460.51,Z 60.126,A -85,B 0,C 180,E1 -8146.626,E2 -8146.626} C_VEL
LIN {X 0,Y 460.536,Z 60.115,A -85,B 0,C 180,E1 -8149.732,E2 -8149.732} C_VEL
LIN {X 0,Y 460.498,Z 60.126,A -85,B 0,C 180,E1 -8152.525,E2 -8152.525} C_VEL
LIN {X 0,Y 460.547,Z 60.114,A -85,B 0,C 180,E1 -8155.624,E2 -8155.624} C_VEL
LIN {X 0,Y 460.54,Z 60.116,A -85,B 0,C 180,E1 -8158.745,E2 -8158.745} C_VEL
LIN {X 0,Y 460.553,Z 60.118,A -85,B 0,C 180,E1 -8162.262,E2 -8162.262} C_VEL
LIN {X 0,Y 460.525,Z 60.117,A -85,B 0,C 180,E1 -8164.704,E2 -8164.704} C_VEL
LIN {X 0,Y 460.514,Z 60.12,A -85,B 0,C 180,E1 -8167.572,E2 -8167.572} C_VEL
LIN {X 0,Y 460.57,Z 60.112,A -85,B 0,C 180,E1 -8170.385,E2 -8170.385} C_VEL
LIN {X 0,Y 460.609,Z 60.113,A -85,B 0,C 180,E1 -8174.059,E2 -8174.059} C_VEL
LIN {X 0,Y 460.581,Z 60.149,A -85,B 0,C 180,E1 -8176.657,E2 -8176.657} C_VEL
LIN {X 0,Y 461.411,Z 65.177,A -85,B 0,C 180,E1 -8177.799,E2 -8177.799} C_VEL
LIN {X 0,Y 461.089,Z 68.342,A -85,B 0,C 180,E1 -8178.391,E2 -8178.391} C_VEL
LIN {X 0,Y 459.865,Z 72.129,A -85,B 0,C 180,E1 -8178.913,E2 -8178.913} C_VEL
LIN {X 0,Y 457.919,Z 77.968,A -85,B 0,C 180,E1 -8179.485,E2 -8179.485} C_VEL
LIN {X 0,Y 456.939,Z 82.941,A -85,B 0,C 180,E1 -8179.807,E2 -8179.807} C_VEL
LIN {X 0,Y 456.933,Z 87.405,A -85,B 0,C 180,E1 -8179.984,E2 -8179.984} C_VEL
LIN {X 0,Y 457.061,Z 88.317,A -85,B 0,C 180,E1 -8180.006,E2 -8180.006} C_VEL
LIN {X 0,Y 457.502,Z 92.427,A -85,B 0,C 180,E1 -8180.087,E2 -8180.087} C_VEL
LIN {X 0,Y 456.657,Z 182.057,A -85,B 0,C 180,E1 -8181.51,E2 -8181.51} C_VEL
LIN {X 0,Y 456.428,Z 195.18,A -85,B 0,C 180,E1 -8181.895,E2 -8181.895} C_VEL
LIN {X 0,Y 456.032,Z 208.356,A -85,B 0,C 180,E1 -8182.473,E2 -8182.473} C_VEL
LIN {X 0,Y 455.756,Z 219.408,A -85,B 0,C 180,E1 -8183.136,E2 -8183.136} C_VEL
LIN {X 0,Y 455.171,Z 230.913,A -85,B 0,C 180,E1 -8184.018,E2 -8184.018} C_VEL
LIN {X 0,Y 454.674,Z 241.254,A -85,B 0,C 180,E1 -8185.012,E2 -8185.012} C_VEL
LIN {X 0,Y 454.245,Z 249.719,A -85,B 0,C 180,E1 -8186.008,E2 -8186.008} C_VEL
LIN {X 0,Y 453.789,Z 257.538,A -85,B 0,C 180,E1 -8187.115,E2 -8187.115} C_VEL
LIN {X 0,Y 453.382,Z 265.192,A -85,B 0,C 180,E1 -8188.446,E2 -8188.446} C_VEL
LIN {X 0,Y 452.955,Z 272.234,A -85,B 0,C 180,E1 -8190,E2 -8190} C_VEL
LIN {X 0,Y 452.734,Z 276.933,A -85,B 0,C 180,E1 -8191.335,E2 -8191.335} C_VEL
LIN {X 0,Y 452.679,Z 280.531,A -85,B 0,C 180,E1 -8192.67,E2 -8192.67} C_VEL
LIN {X 0,Y 452.641,Z 282.396,A -85,B 0,C 180,E1 -8193.561,E2 -8193.561} C_VEL
LIN {X 0,Y 452.518,Z 283.811,A -85,B 0,C 180,E1 -8194.454,E2 -8194.454} C_VEL
LIN {X 0,Y 452.587,Z 285.428,A -85,B 0,C 180,E1 -8196.241,E2 -8196.241} C_VEL
LIN {X 0,Y 452.549,Z 285.668,A -85,B 0,C 180,E1 -8197.137,E2 -8197.137} C_VEL
LIN {X 0,Y 452.515,Z 285.477,A -85,B 0,C 180,E1 -8198.035,E2 -8198.035} C_VEL
LIN {X 0,Y 452.498,Z 283.908,A -85,B 0,C 180,E1 -8199.837,E2 -8199.837} C_VEL
LIN {X 0,Y 452.615,Z 282.524,A -85,B 0,C 180,E1 -8200.739,E2 -8200.739} C_VEL
LIN {X 0,Y 452.794,Z 279.637,A -85,B 0,C 180,E1 -8202.08,E2 -8202.08} C_VEL
LIN {X 0,Y 452.979,Z 275.614,A -85,B 0,C 180,E1 -8203.458,E2 -8203.458} C_VEL
LIN {X 0,Y 453.395,Z 269.427,A -85,B 0,C 180,E1 -8205.049,E2 -8205.049} C_VEL
LIN {X 0,Y 453.775,Z 262.64,A -85,B 0,C 180,E1 -8206.419,E2 -8206.419} C_VEL
LIN {X 0,Y 454.235,Z 254.145,A -85,B 0,C 180,E1 -8207.793,E2 -8207.793} C_VEL
LIN {X 0,Y 454.901,Z 243.94,A -85,B 0,C 180,E1 -8209.097,E2 -8209.097} C_VEL
LIN {X 0,Y 455.434,Z 234.426,A -85,B 0,C 180,E1 -8210.081,E2 -8210.081} C_VEL
LIN {X 0,Y 456.034,Z 223.43,A -85,B 0,C 180,E1 -8210.997,E2 -8210.997} C_VEL
LIN {X 0,Y 456.568,Z 210.996,A -85,B 0,C 180,E1 -8211.8,E2 -8211.8} C_VEL
LIN {X 0,Y 457.032,Z 199.186,A -85,B 0,C 180,E1 -8212.371,E2 -8212.371} C_VEL
LIN {X 0,Y 457.379,Z 187.008,A -85,B 0,C 180,E1 -8212.786,E2 -8212.786} C_VEL
LIN {X 0,Y 457.543,Z 172.526,A -85,B 0,C 180,E1 -8213.079,E2 -8213.079} C_VEL
LIN {X 0,Y 458.317,Z 90.359,A -85,B 0,C 180,E1 -8214.382,E2 -8214.382} C_VEL
LIN {X 0,Y 454.911,Z 75.566,A -85,B 0,C 180,E1 -8214.784,E2 -8214.784} C_VEL
LIN {X 0,Y 454.899,Z 68.573,A -85,B 0,C 180,E1 -8216.352,E2 -8216.352} C_VEL
LIN {X 0,Y 453.51,Z 60.995,A -85,B 0,C 180,E1 -8218.187,E2 -8218.187} C_VEL
LIN {X 0,Y 453.443,Z 61.002,A -85,B 0,C 180,E1 -8221.519,E2 -8221.519} C_VEL
LIN {X 0,Y 453.475,Z 60.997,A -85,B 0,C 180,E1 -8224.774,E2 -8224.774} C_VEL
LIN {X 0,Y 453.443,Z 61.005,A -85,B 0,C 180,E1 -8228.314,E2 -8228.314} C_VEL
LIN {X 0,Y 453.47,Z 60.997,A -85,B 0,C 180,E1 -8230.612,E2 -8230.612} C_VEL
LIN {X 0,Y 453.479,Z 60.986,A -85,B 0,C 180,E1 -8234.527,E2 -8234.527} C_VEL
LIN {X 0,Y 453.434,Z 61.001,A -85,B 0,C 180,E1 -8238.072,E2 -8238.072} C_VEL
LIN {X 0,Y 453.424,Z 61.002,A -85,B 0,C 180,E1 -8240.805,E2 -8240.805} C_VEL
LIN {X 0,Y 453.439,Z 60.999,A -85,B 0,C 180,E1 -8243.915,E2 -8243.915} C_VEL
LIN {X 0,Y 453.468,Z 60.998,A -85,B 0,C 180,E1 -8246.816,E2 -8246.816} C_VEL
LIN {X 0,Y 453.45,Z 60.998,A -85,B 0,C 180,E1 -8250.266,E2 -8250.266} C_VEL
LIN {X 0,Y 453.426,Z 61.004,A -85,B 0,C 180,E1 -8253.288,E2 -8253.288} C_VEL
LIN {X 0,Y 453.493,Z 60.992,A -85,B 0,C 180,E1 -8256.238,E2 -8256.238} C_VEL
LIN {X 0,Y 453.485,Z 60.999,A -85,B 0,C 180,E1 -8259.117,E2 -8259.117} C_VEL
LIN {X 0,Y 453.502,Z 60.987,A -85,B 0,C 180,E1 -8261.944,E2 -8261.944} C_VEL
LIN {X 0,Y 453.533,Z 60.994,A -85,B 0,C 180,E1 -8264.726,E2 -8264.726} C_VEL
LIN {X 0,Y 453.56,Z 60.982,A -85,B 0,C 180,E1 -8268.379,E2 -8268.379} C_VEL
LIN {X 0,Y 453.58,Z 60.983,A -85,B 0,C 180,E1 -8271.086,E2 -8271.086} C_VEL
LIN {X 0,Y 453.631,Z 60.97,A -85,B 0,C 180,E1 -8273.774,E2 -8273.774} C_VEL
LIN {X 0,Y 453.717,Z 60.964,A -85,B 0,C 180,E1 -8277.336,E2 -8277.336} C_VEL
LIN {X 0,Y 453.77,Z 60.956,A -85,B 0,C 180,E1 -8280,E2 -8280} C_VEL
LIN {X 0,Y 453.707,Z 60.967,A -85,B 0,C 180,E1 -8282.663,E2 -8282.663} C_VEL
LIN {X 0,Y 453.64,Z 60.973,A -85,B 0,C 180,E1 -8286.226,E2 -8286.226} C_VEL
LIN {X 0,Y 453.581,Z 60.981,A -85,B 0,C 180,E1 -8288.913,E2 -8288.913} C_VEL
LIN {X 0,Y 453.567,Z 60.98,A -85,B 0,C 180,E1 -8292.529,E2 -8292.529} C_VEL
LIN {X 0,Y 453.54,Z 60.983,A -85,B 0,C 180,E1 -8296.196,E2 -8296.196} C_VEL
LIN {X 0,Y 453.519,Z 60.989,A -85,B 0,C 180,E1 -8299.039,E2 -8299.039} C_VEL
LIN {X 0,Y 453.479,Z 60.991,A -85,B 0,C 180,E1 -8301.836,E2 -8301.836} C_VEL
LIN {X 0,Y 453.495,Z 60.994,A -85,B 0,C 180,E1 -8304.735,E2 -8304.735} C_VEL
LIN {X 0,Y 453.531,Z 60.988,A -85,B 0,C 180,E1 -8307.959,E2 -8307.959} C_VEL
LIN {X 0,Y 453.468,Z 60.997,A -85,B 0,C 180,E1 -8311.525,E2 -8311.525} C_VEL
LIN {X 0,Y 453.49,Z 60.993,A -85,B 0,C 180,E1 -8314.777,E2 -8314.777} C_VEL
LIN {X 0,Y 453.465,Z 60.993,A -85,B 0,C 180,E1 -8318.312,E2 -8318.312} C_VEL
LIN {X 0,Y 453.496,Z 60.997,A -85,B 0,C 180,E1 -8320.609,E2 -8320.609} C_VEL
LIN {X 0,Y 453.457,Z 60.999,A -85,B 0,C 180,E1 -8323.244,E2 -8323.244} C_VEL
LIN {X 0,Y 453.466,Z 60.996,A -85,B 0,C 180,E1 -8325.779,E2 -8325.779} C_VEL
LIN {X 0,Y 453.482,Z 60.997,A -85,B 0,C 180,E1 -8328.209,E2 -8328.209} C_VEL
LIN {X 0,Y 453.518,Z 60.992,A -85,B 0,C 180,E1 -8330.79,E2 -8330.79} C_VEL
LIN {X 0,Y 453.457,Z 61.001,A -85,B 0,C 180,E1 -8333.917,E2 -8333.917} C_VEL
LIN {X 0,Y 453.486,Z 60.998,A -85,B 0,C 180,E1 -8337.151,E2 -8337.151} C_VEL
LIN {X 0,Y 453.477,Z 61.003,A -85,B 0,C 180,E1 -8340.268,E2 -8340.268} C_VEL
LIN {X 0,Y 453.563,Z 61.024,A -85,B 0,C 180,E1 -8342.737,E2 -8342.737} C_VEL
LIN {X 0,Y 456.224,Z 74.253,A -85,B 0,C 180,E1 -8345.351,E2 -8345.351} C_VEL
LIN {X 0,Y 456.114,Z 79.945,A -85,B 0,C 180,E1 -8346.383,E2 -8346.383} C_VEL
LIN {X 0,Y 455.146,Z 97.167,A -85,B 0,C 180,E1 -8349.434,E2 -8349.434} C_VEL
LIN {X 0,Y 454.444,Z 113.073,A -85,B 0,C 180,E1 -8352.218,E2 -8352.218} C_VEL
LIN {X 0,Y 457.899,Z 135.345,A -85,B 0,C 180,E1 -8352.751,E2 -8352.751} C_VEL
LIN {X 0,Y 457.206,Z 221.478,A -85,B 0,C 180,E1 -8354.137,E2 -8354.137} C_VEL
LIN {X 0,Y 456.743,Z 234.831,A -85,B 0,C 180,E1 -8354.521,E2 -8354.521} C_VEL
LIN {X 0,Y 456.157,Z 248.152,A -85,B 0,C 180,E1 -8355.101,E2 -8355.101} C_VEL
LIN {X 0,Y 455.527,Z 260.135,A -85,B 0,C 180,E1 -8355.822,E2 -8355.822} C_VEL
LIN {X 0,Y 454.815,Z 272.407,A -85,B 0,C 180,E1 -8356.782,E2 -8356.782} C_VEL
LIN {X 0,Y 454.317,Z 281.962,A -85,B 0,C 180,E1 -8357.719,E2 -8357.719} C_VEL
LIN {X 0,Y 453.758,Z 291.289,A -85,B 0,C 180,E1 -8358.836,E2 -8358.836} C_VEL
LIN {X 0,Y 453.291,Z 298.976,A -85,B 0,C 180,E1 -8359.955,E2 -8359.955} C_VEL
LIN {X 0,Y 452.939,Z 306.522,A -85,B 0,C 180,E1 -8361.298,E2 -8361.298} C_VEL
LIN {X 0,Y 452.663,Z 313.514,A -85,B 0,C 180,E1 -8362.865,E2 -8362.865} C_VEL
LIN {X 0,Y 452.512,Z 318.145,A -85,B 0,C 180,E1 -8364.206,E2 -8364.206} C_VEL
LIN {X 0,Y 452.485,Z 321.679,A -85,B 0,C 180,E1 -8365.546,E2 -8365.546} C_VEL
LIN {X 0,Y 452.491,Z 323.473,A -85,B 0,C 180,E1 -8366.438,E2 -8366.438} C_VEL
LIN {X 0,Y 452.527,Z 324.835,A -85,B 0,C 180,E1 -8367.329,E2 -8367.329} C_VEL
LIN {X 0,Y 452.497,Z 326.377,A -85,B 0,C 180,E1 -8369.11,E2 -8369.11} C_VEL
LIN {X 0,Y 452.478,Z 326.528,A -85,B 0,C 180,E1 -8370,E2 -8370} C_VEL
LIN {X 0,Y 452.497,Z 326.271,A -85,B 0,C 180,E1 -8370.89,E2 -8370.89} C_VEL
LIN {X 0,Y 452.53,Z 324.592,A -85,B 0,C 180,E1 -8372.67,E2 -8372.67} C_VEL
LIN {X 0,Y 452.521,Z 323.116,A -85,B 0,C 180,E1 -8373.561,E2 -8373.561} C_VEL
LIN {X 0,Y 452.543,Z 320.093,A -85,B 0,C 180,E1 -8374.9,E2 -8374.9} C_VEL
LIN {X 0,Y 452.514,Z 315.834,A -85,B 0,C 180,E1 -8376.286,E2 -8376.286} C_VEL
LIN {X 0,Y 452.748,Z 309.718,A -85,B 0,C 180,E1 -8377.806,E2 -8377.806} C_VEL
LIN {X 0,Y 452.998,Z 302.871,A -85,B 0,C 180,E1 -8379.15,E2 -8379.15} C_VEL
LIN {X 0,Y 453.328,Z 294.342,A -85,B 0,C 180,E1 -8380.495,E2 -8380.495} C_VEL
LIN {X 0,Y 453.855,Z 285.566,A -85,B 0,C 180,E1 -8381.613,E2 -8381.613} C_VEL
LIN {X 0,Y 454.361,Z 275.303,A -85,B 0,C 180,E1 -8382.68,E2 -8382.68} C_VEL
LIN {X 0,Y 454.889,Z 263.96,A -85,B 0,C 180,E1 -8383.627,E2 -8383.627} C_VEL
LIN {X 0,Y 455.49,Z 251.846,A -85,B 0,C 180,E1 -8384.406,E2 -8384.406} C_VEL
LIN {X 0,Y 455.989,Z 239.199,A -85,B 0,C 180,E1 -8385.018,E2 -8385.018} C_VEL
LIN {X 0,Y 456.404,Z 226.929,A -85,B 0,C 180,E1 -8385.433,E2 -8385.433} C_VEL
LIN {X 0,Y 456.592,Z 213.096,A -85,B 0,C 180,E1 -8385.712,E2 -8385.712} C_VEL
LIN {X 0,Y 457.057,Z 134.191,A -85,B 0,C 180,E1 -8386.953,E2 -8386.953} C_VEL
LIN {X 0,Y 454.174,Z 113.234,A -85,B 0,C 180,E1 -8387.411,E2 -8387.411} C_VEL
LIN {X 0,Y 454.842,Z 94.798,A -85,B 0,C 180,E1 -8390.58,E2 -8390.58} C_VEL
LIN {X 0,Y 455.779,Z 75.814,A -85,B 0,C 180,E1 -8393.872,E2 -8393.872} C_VEL
LIN {X 0,Y 455.617,Z 71.677,A -85,B 0,C 180,E1 -8394.612,E2 -8394.612} C_VEL
LIN {X 0,Y 453.56,Z 60.99,A -85,B 0,C 180,E1 -8396.66,E2 -8396.66} C_VEL
LIN {X 0,Y 453.473,Z 61.001,A -85,B 0,C 180,E1 -8399.785,E2 -8399.785} C_VEL
LIN {X 0,Y 453.491,Z 60.993,A -85,B 0,C 180,E1 -8403.189,E2 -8403.189} C_VEL
LIN {X 0,Y 453.453,Z 60.999,A -85,B 0,C 180,E1 -8406.299,E2 -8406.299} C_VEL
LIN {X 0,Y 453.517,Z 60.993,A -85,B 0,C 180,E1 -8409.447,E2 -8409.447} C_VEL
LIN {X 0,Y 453.462,Z 60.997,A -85,B 0,C 180,E1 -8412.995,E2 -8412.995} C_VEL
LIN {X 0,Y 453.463,Z 60.999,A -85,B 0,C 180,E1 -8415.779,E2 -8415.779} C_VEL
LIN {X 0,Y 453.478,Z 60.994,A -85,B 0,C 180,E1 -8418.209,E2 -8418.209} C_VEL
LIN {X 0,Y 453.491,Z 60.994,A -85,B 0,C 180,E1 -8420.794,E2 -8420.794} C_VEL
LIN {X 0,Y 453.454,Z 60.997,A -85,B 0,C 180,E1 -8423.917,E2 -8423.917} C_VEL
LIN {X 0,Y 453.482,Z 61.001,A -85,B 0,C 180,E1 -8427.151,E2 -8427.151} C_VEL
LIN {X 0,Y 453.474,Z 60.994,A -85,B 0,C 180,E1 -8430.268,E2 -8430.268} C_VEL
LIN {X 0,Y 453.506,Z 60.993,A -85,B 0,C 180,E1 -8433.294,E2 -8433.294} C_VEL
LIN {X 0,Y 453.501,Z 60.992,A -85,B 0,C 180,E1 -8436.239,E2 -8436.239} C_VEL
LIN {X 0,Y 453.482,Z 60.996,A -85,B 0,C 180,E1 -8439.118,E2 -8439.118} C_VEL
LIN {X 0,Y 453.503,Z 60.991,A -85,B 0,C 180,E1 -8441.944,E2 -8441.944} C_VEL
LIN {X 0,Y 453.539,Z 60.992,A -85,B 0,C 180,E1 -8444.726,E2 -8444.726} C_VEL
LIN {X 0,Y 453.558,Z 60.99,A -85,B 0,C 180,E1 -8448.379,E2 -8448.379} C_VEL
LIN {X 0,Y 453.651,Z 60.975,A -85,B 0,C 180,E1 -8451.985,E2 -8451.985} C_VEL
LIN {X 0,Y 453.667,Z 60.973,A -85,B 0,C 180,E1 -8454.667,E2 -8454.667} C_VEL
LIN {X 0,Y 453.736,Z 60.962,A -85,B 0,C 180,E1 -8457.337,E2 -8457.337} C_VEL
LIN {X 0,Y 453.821,Z 60.957,A -85,B 0,C 180,E1 -8460,E2 -8460} C_VEL
LIN {X 0,Y 453.736,Z 60.962,A -85,B 0,C 180,E1 -8462.664,E2 -8462.664} C_VEL
LIN {X 0,Y 453.651,Z 60.976,A -85,B 0,C 180,E1 -8466.226,E2 -8466.226} C_VEL
LIN {X 0,Y 453.585,Z 60.98,A -85,B 0,C 180,E1 -8468.914,E2 -8468.914} C_VEL
LIN {X 0,Y 453.564,Z 60.983,A -85,B 0,C 180,E1 -8472.529,E2 -8472.529} C_VEL
LIN {X 0,Y 453.544,Z 60.986,A -85,B 0,C 180,E1 -8476.196,E2 -8476.196} C_VEL
LIN {X 0,Y 453.516,Z 60.991,A -85,B 0,C 180,E1 -8479.039,E2 -8479.039} C_VEL
LIN {X 0,Y 453.477,Z 60.996,A -85,B 0,C 180,E1 -8481.836,E2 -8481.836} C_VEL
LIN {X 0,Y 453.492,Z 60.993,A -85,B 0,C 180,E1 -8484.736,E2 -8484.736} C_VEL
LIN {X 0,Y 453.529,Z 60.988,A -85,B 0,C 180,E1 -8487.959,E2 -8487.959} C_VEL
LIN {X 0,Y 453.465,Z 60.998,A -85,B 0,C 180,E1 -8491.525,E2 -8491.525} C_VEL
LIN {X 0,Y 453.483,Z 60.998,A -85,B 0,C 180,E1 -8494.777,E2 -8494.777} C_VEL
LIN {X 0,Y 453.459,Z 60.997,A -85,B 0,C 180,E1 -8498.313,E2 -8498.313} C_VEL
LIN {X 0,Y 453.471,Z 61,A -85,B 0,C 180,E1 -8500.612,E2 -8500.612} C_VEL
LIN {X 0,Y 453.46,Z 60.998,A -85,B 0,C 180,E1 -8504.222,E2 -8504.222} C_VEL
LIN {X 0,Y 453.45,Z 61,A -85,B 0,C 180,E1 -8507.004,E2 -8507.004} C_VEL
LIN {X 0,Y 453.495,Z 60.991,A -85,B 0,C 180,E1 -8509.41,E2 -8509.41} C_VEL
LIN {X 0,Y 453.45,Z 61,A -85,B 0,C 180,E1 -8512.81,E2 -8512.81} C_VEL
LIN {X 0,Y 453.478,Z 60.998,A -85,B 0,C 180,E1 -8516.088,E2 -8516.088} C_VEL
LIN {X 0,Y 453.478,Z 60.993,A -85,B 0,C 180,E1 -8519.241,E2 -8519.241} C_VEL
LIN {X 0,Y 453.51,Z 60.995,A -85,B 0,C 180,E1 -8522.296,E2 -8522.296} C_VEL
LIN {X 0,Y 453.473,Z 60.995,A -85,B 0,C 180,E1 -8525.263,E2 -8525.263} C_VEL
LIN {X 0,Y 453.484,Z 60.995,A -85,B 0,C 180,E1 -8528.415,E2 -8528.415} C_VEL
LIN {X 0,Y 453.526,Z 60.988,A -85,B 0,C 180,E1 -8531.009,E2 -8531.009} C_VEL
LIN {X 0,Y 453.573,Z 60.992,A -85,B 0,C 180,E1 -8533.88,E2 -8533.88} C_VEL
LIN {X 0,Y 453.555,Z 61.017,A -85,B 0,C 180,E1 -8536.503,E2 -8536.503} C_VEL
LIN {X 0,Y 454.636,Z 68.363,A -85,B 0,C 180,E1 -8538.181,E2 -8538.181} C_VEL
LIN {X 0,Y 454.567,Z 75.366,A -85,B 0,C 180,E1 -8539.709,E2 -8539.709} C_VEL
LIN {X 0,Y 457.061,Z 88.317,A -85,B 0,C 180,E1 -8540.006,E2 -8540.006} C_VEL
LIN {X 0,Y 457.262,Z 92.173,A -85,B 0,C 180,E1 -8540.075,E2 -8540.075} C_VEL
LIN {X 0,Y 456.312,Z 97.97,A -85,B 0,C 180,E1 -8540.135,E2 -8540.135} C_VEL
LIN {X 0,Y 451.312,Z 113.217,A -85,B 0,C 180,E1 -8540.208,E2 -8540.208} C_VEL
LIN {X 0,Y 450.422,Z 119.132,A -85,B 0,C 180,E1 -8540.273,E2 -8540.273} C_VEL
LIN {X 0,Y 449.782,Z 182.26,A -85,B 0,C 180,E1 -8541.294,E2 -8541.294} C_VEL
LIN {X 0,Y 449.554,Z 195.42,A -85,B 0,C 180,E1 -8541.686,E2 -8541.686} C_VEL
LIN {X 0,Y 449.151,Z 208.065,A -85,B 0,C 180,E1 -8542.244,E2 -8542.244} C_VEL
LIN {X 0,Y 448.867,Z 219.285,A -85,B 0,C 180,E1 -8542.918,E2 -8542.918} C_VEL
LIN {X 0,Y 448.245,Z 230.886,A -85,B 0,C 180,E1 -8543.812,E2 -8543.812} C_VEL
LIN {X 0,Y 447.738,Z 241.287,A -85,B 0,C 180,E1 -8544.822,E2 -8544.822} C_VEL
LIN {X 0,Y 447.21,Z 250.683,A -85,B 0,C 180,E1 -8545.945,E2 -8545.945} C_VEL
LIN {X 0,Y 446.632,Z 259.736,A -85,B 0,C 180,E1 -8547.295,E2 -8547.295} C_VEL
LIN {X 0,Y 446.273,Z 267.022,A -85,B 0,C 180,E1 -8548.647,E2 -8548.647} C_VEL
LIN {X 0,Y 445.874,Z 272.886,A -85,B 0,C 180,E1 -8550,E2 -8550} C_VEL
LIN {X 0,Y 445.652,Z 277.514,A -85,B 0,C 180,E1 -8551.356,E2 -8551.356} C_VEL
LIN {X 0,Y 445.594,Z 281.047,A -85,B 0,C 180,E1 -8552.712,E2 -8552.712} C_VEL
LIN {X 0,Y 445.551,Z 282.867,A -85,B 0,C 180,E1 -8553.618,E2 -8553.618} C_VEL
LIN {X 0,Y 445.476,Z 285.205,A -85,B 0,C 180,E1 -8555.432,E2 -8555.432} C_VEL
LIN {X 0,Y 445.532,Z 285.817,A -85,B 0,C 180,E1 -8556.386,E2 -8556.386} C_VEL
LIN {X 0,Y 445.459,Z 285.987,A -85,B 0,C 180,E1 -8557.251,E2 -8557.251} C_VEL
LIN {X 0,Y 445.418,Z 285.134,A -85,B 0,C 180,E1 -8559.079,E2 -8559.079} C_VEL
LIN {X 0,Y 445.425,Z 284.126,A -85,B 0,C 180,E1 -8559.995,E2 -8559.995} C_VEL
LIN {X 0,Y 445.556,Z 282.686,A -85,B 0,C 180,E1 -8560.911,E2 -8560.911} C_VEL
LIN {X 0,Y 445.73,Z 280.042,A -85,B 0,C 180,E1 -8562.153,E2 -8562.153} C_VEL
LIN {X 0,Y 445.954,Z 275.649,A -85,B 0,C 180,E1 -8563.674,E2 -8563.674} C_VEL
LIN {X 0,Y 446.38,Z 269.374,A -85,B 0,C 180,E1 -8565.291,E2 -8565.291} C_VEL
LIN {X 0,Y 446.809,Z 262.505,A -85,B 0,C 180,E1 -8566.682,E2 -8566.682} C_VEL
LIN {X 0,Y 447.22,Z 255.452,A -85,B 0,C 180,E1 -8567.845,E2 -8567.845} C_VEL
LIN {X 0,Y 447.846,Z 246.908,A -85,B 0,C 180,E1 -8569.004,E2 -8569.004} C_VEL
LIN {X 0,Y 448.446,Z 236.264,A -85,B 0,C 180,E1 -8570.169,E2 -8570.169} C_VEL
LIN {X 0,Y 449.047,Z 225.661,A -85,B 0,C 180,E1 -8571.099,E2 -8571.099} C_VEL
LIN {X 0,Y 449.688,Z 213.904,A -85,B 0,C 180,E1 -8571.909,E2 -8571.909} C_VEL
LIN {X 0,Y 450.21,Z 201.576,A -85,B 0,C 180,E1 -8572.547,E2 -8572.547} C_VEL
LIN {X 0,Y 450.605,Z 189.081,A -85,B 0,C 180,E1 -8573.006,E2 -8573.006} C_VEL
LIN {X 0,Y 450.77,Z 175.285,A -85,B 0,C 180,E1 -8573.318,E2 -8573.318} C_VEL
LIN {X 0,Y 451.579,Z 91.254,A -85,B 0,C 180,E1 -8574.672,E2 -8574.672} C_VEL
LIN {X 0,Y 448.024,Z 75.787,A -85,B 0,C 180,E1 -8575.121,E2 -8575.121} C_VEL
LIN {X 0,Y 447.98,Z 70.036,A -85,B 0,C 180,E1 -8576.429,E2 -8576.429} C_VEL
LIN {X 0,Y 446.473,Z 61.872,A -85,B 0,C 180,E1 -8578.41,E2 -8578.41} C_VEL
LIN {X 0,Y 446.395,Z 61.882,A -85,B 0,C 180,E1 -8581.769,E2 -8581.769} C_VEL
LIN {X 0,Y 446.415,Z 61.877,A -85,B 0,C 180,E1 -8584.525,E2 -8584.525} C_VEL
LIN {X 0,Y 446.391,Z 61.879,A -85,B 0,C 180,E1 -8587.881,E2 -8587.881} C_VEL
LIN {X 0,Y 446.399,Z 61.877,A -85,B 0,C 180,E1 -8590.913,E2 -8590.913} C_VEL
LIN {X 0,Y 446.385,Z 61.877,A -85,B 0,C 180,E1 -8593.848,E2 -8593.848} C_VEL
LIN {X 0,Y 446.386,Z 61.879,A -85,B 0,C 180,E1 -8596.406,E2 -8596.406} C_VEL
LIN {X 0,Y 446.391,Z 61.883,A -85,B 0,C 180,E1 -8599.796,E2 -8599.796} C_VEL
LIN {X 0,Y 446.391,Z 61.882,A -85,B 0,C 180,E1 -8603.253,E2 -8603.253} C_VEL
LIN {X 0,Y 446.427,Z 61.873,A -85,B 0,C 180,E1 -8606.551,E2 -8606.551} C_VEL
LIN {X 0,Y 446.417,Z 61.875,A -85,B 0,C 180,E1 -8609.983,E2 -8609.983} C_VEL
LIN {X 0,Y 446.385,Z 61.878,A -85,B 0,C 180,E1 -8612.833,E2 -8612.833} C_VEL
LIN {X 0,Y 446.426,Z 61.872,A -85,B 0,C 180,E1 -8615.936,E2 -8615.936} C_VEL
LIN {X 0,Y 446.457,Z 61.871,A -85,B 0,C 180,E1 -8618.773,E2 -8618.773} C_VEL
LIN {X 0,Y 446.452,Z 61.866,A -85,B 0,C 180,E1 -8621.649,E2 -8621.649} C_VEL
LIN {X 0,Y 446.48,Z 61.869,A -85,B 0,C 180,E1 -8624.478,E2 -8624.478} C_VEL
LIN {X 0,Y 446.519,Z 61.858,A -85,B 0,C 180,E1 -8628.193,E2 -8628.193} C_VEL
LIN {X 0,Y 446.528,Z 61.862,A -85,B 0,C 180,E1 -8630.944,E2 -8630.944} C_VEL
LIN {X 0,Y 446.602,Z 61.845,A -85,B 0,C 180,E1 -8633.675,E2 -8633.675} C_VEL
LIN {X 0,Y 446.667,Z 61.843,A -85,B 0,C 180,E1 -8637.294,E2 -8637.294} C_VEL
LIN {X 0,Y 446.721,Z 61.834,A -85,B 0,C 180,E1 -8640,E2 -8640} C_VEL
LIN {X 0,Y 446.657,Z 61.845,A -85,B 0,C 180,E1 -8642.705,E2 -8642.705} C_VEL
LIN {X 0,Y 446.609,Z 61.849,A -85,B 0,C 180,E1 -8646.324,E2 -8646.324} C_VEL
LIN {X 0,Y 446.529,Z 61.86,A -85,B 0,C 180,E1 -8649.055,E2 -8649.055} C_VEL
LIN {X 0,Y 446.525,Z 61.856,A -85,B 0,C 180,E1 -8652.73,E2 -8652.73} C_VEL
LIN {X 0,Y 446.487,Z 61.86,A -85,B 0,C 180,E1 -8656.459,E2 -8656.459} C_VEL
LIN {X 0,Y 446.471,Z 61.87,A -85,B 0,C 180,E1 -8659.303,E2 -8659.303} C_VEL
LIN {X 0,Y 446.42,Z 61.868,A -85,B 0,C 180,E1 -8662.199,E2 -8662.199} C_VEL
LIN {X 0,Y 446.439,Z 61.877,A -85,B 0,C 180,E1 -8665.153,E2 -8665.153} C_VEL
LIN {X 0,Y 446.488,Z 61.865,A -85,B 0,C 180,E1 -8668.178,E2 -8668.178} C_VEL
LIN {X 0,Y 446.421,Z 61.873,A -85,B 0,C 180,E1 -8671.775,E2 -8671.775} C_VEL
LIN {X 0,Y 446.432,Z 61.874,A -85,B 0,C 180,E1 -8674.523,E2 -8674.523} C_VEL
LIN {X 0,Y 446.417,Z 61.87,A -85,B 0,C 180,E1 -8678.079,E2 -8678.079} C_VEL
LIN {X 0,Y 446.429,Z 61.876,A -85,B 0,C 180,E1 -8680.917,E2 -8680.917} C_VEL
LIN {X 0,Y 446.402,Z 61.877,A -85,B 0,C 180,E1 -8683.846,E2 -8683.846} C_VEL
LIN {X 0,Y 446.401,Z 61.879,A -85,B 0,C 180,E1 -8686.403,E2 -8686.403} C_VEL
LIN {X 0,Y 446.43,Z 61.873,A -85,B 0,C 180,E1 -8689.082,E2 -8689.082} C_VEL
LIN {X 0,Y 446.418,Z 61.876,A -85,B 0,C 180,E1 -8691.92,E2 -8691.92} C_VEL
LIN {X 0,Y 446.431,Z 61.874,A -85,B 0,C 180,E1 -8695.477,E2 -8695.477} C_VEL
LIN {X 0,Y 446.419,Z 61.88,A -85,B 0,C 180,E1 -8698.699,E2 -8698.699} C_VEL
LIN {X 0,Y 446.517,Z 61.868,A -85,B 0,C 180,E1 -8702.334,E2 -8702.334} C_VEL
LIN {X 0,Y 446.531,Z 61.929,A -85,B 0,C 180,E1 -8702.462,E2 -8702.462} C_VEL
LIN {X 0,Y 449.257,Z 75.206,A -85,B 0,C 180,E1 -8705.139,E2 -8705.139} C_VEL
LIN {X 0,Y 449.397,Z 78.621,A -85,B 0,C 180,E1 -8705.782,E2 -8705.782} C_VEL
LIN {X 0,Y 448.285,Z 97.043,A -85,B 0,C 180,E1 -8709.104,E2 -8709.104} C_VEL
LIN {X 0,Y 447.506,Z 112.839,A -85,B 0,C 180,E1 -8711.917,E2 -8711.917} C_VEL
LIN {X 0,Y 450.987,Z 134.666,A -85,B 0,C 180,E1 -8712.439,E2 -8712.439} C_VEL
LIN {X 0,Y 451.192,Z 141.692,A -85,B 0,C 180,E1 -8712.565,E2 -8712.565} C_VEL
LIN {X 0,Y 450.444,Z 221.239,A -85,B 0,C 180,E1 -8713.864,E2 -8713.864} C_VEL
LIN {X 0,Y 449.953,Z 234.556,A -85,B 0,C 180,E1 -8714.253,E2 -8714.253} C_VEL
LIN {X 0,Y 449.35,Z 247.299,A -85,B 0,C 180,E1 -8714.812,E2 -8714.812} C_VEL
LIN {X 0,Y 448.766,Z 258.636,A -85,B 0,C 180,E1 -8715.488,E2 -8715.488} C_VEL
LIN {X 0,Y 448.03,Z 270.325,A -85,B 0,C 180,E1 -8716.391,E2 -8716.391} C_VEL
LIN {X 0,Y 447.411,Z 280.842,A -85,B 0,C 180,E1 -8717.411,E2 -8717.411} C_VEL
LIN {X 0,Y 446.901,Z 289.454,A -85,B 0,C 180,E1 -8718.433,E2 -8718.433} C_VEL
LIN {X 0,Y 446.314,Z 297.406,A -85,B 0,C 180,E1 -8719.567,E2 -8719.567} C_VEL
LIN {X 0,Y 445.934,Z 305.214,A -85,B 0,C 180,E1 -8720.932,E2 -8720.932} C_VEL
LIN {X 0,Y 445.667,Z 311.478,A -85,B 0,C 180,E1 -8722.297,E2 -8722.297} C_VEL
LIN {X 0,Y 445.432,Z 317.55,A -85,B 0,C 180,E1 -8724,E2 -8724} C_VEL
LIN {X 0,Y 445.41,Z 321.42,A -85,B 0,C 180,E1 -8725.475,E2 -8725.475} C_VEL
LIN {X 0,Y 445.39,Z 323.194,A -85,B 0,C 180,E1 -8726.381,E2 -8726.381} C_VEL
LIN {X 0,Y 445.45,Z 324.547,A -85,B 0,C 180,E1 -8727.287,E2 -8727.287} C_VEL
LIN {X 0,Y 445.403,Z 326.069,A -85,B 0,C 180,E1 -8729.096,E2 -8729.096} C_VEL
LIN {X 0,Y 445.413,Z 326.203,A -85,B 0,C 180,E1 -8730,E2 -8730} C_VEL
LIN {X 0,Y 445.402,Z 325.282,A -85,B 0,C 180,E1 -8731.808,E2 -8731.808} C_VEL
LIN {X 0,Y 445.455,Z 324.239,A -85,B 0,C 180,E1 -8732.713,E2 -8732.713} C_VEL
LIN {X 0,Y 445.419,Z 322.742,A -85,B 0,C 180,E1 -8733.618,E2 -8733.618} C_VEL
LIN {X 0,Y 445.47,Z 319.699,A -85,B 0,C 180,E1 -8734.978,E2 -8734.978} C_VEL
LIN {X 0,Y 445.45,Z 315.583,A -85,B 0,C 180,E1 -8736.34,E2 -8736.34} C_VEL
LIN {X 0,Y 445.679,Z 309.274,A -85,B 0,C 180,E1 -8737.931,E2 -8737.931} C_VEL
LIN {X 0,Y 445.933,Z 302.397,A -85,B 0,C 180,E1 -8739.296,E2 -8739.296} C_VEL
LIN {X 0,Y 446.309,Z 293.818,A -85,B 0,C 180,E1 -8740.662,E2 -8740.662} C_VEL
LIN {X 0,Y 446.83,Z 284.996,A -85,B 0,C 180,E1 -8741.798,E2 -8741.798} C_VEL
LIN {X 0,Y 447.415,Z 273.891,A -85,B 0,C 180,E1 -8742.957,E2 -8742.957} C_VEL
LIN {X 0,Y 447.94,Z 263.241,A -85,B 0,C 180,E1 -8743.843,E2 -8743.843} C_VEL
LIN {X 0,Y 448.56,Z 251.01,A -85,B 0,C 180,E1 -8744.634,E2 -8744.634} C_VEL
LIN {X 0,Y 449.112,Z 238.204,A -85,B 0,C 180,E1 -8745.253,E2 -8745.253} C_VEL
LIN {X 0,Y 449.544,Z 225.443,A -85,B 0,C 180,E1 -8745.674,E2 -8745.674} C_VEL
LIN {X 0,Y 449.83,Z 207.33,A -85,B 0,C 180,E1 -8746.013,E2 -8746.013} C_VEL
LIN {X 0,Y 450.203,Z 135.138,A -85,B 0,C 180,E1 -8747.167,E2 -8747.167} C_VEL
LIN {X 0,Y 447.162,Z 112.916,A -85,B 0,C 180,E1 -8747.66,E2 -8747.66} C_VEL
LIN {X 0,Y 447.844,Z 95.645,A -85,B 0,C 180,E1 -8750.676,E2 -8750.676} C_VEL
LIN {X 0,Y 448.846,Z 76.644,A -85,B 0,C 180,E1 -8754.023,E2 -8754.023} C_VEL
LIN {X 0,Y 448.659,Z 72.957,A -85,B 0,C 180,E1 -8754.696,E2 -8754.696} C_VEL
LIN {X 0,Y 446.524,Z 61.866,A -85,B 0,C 180,E1 -8756.867,E2 -8756.867} C_VEL
LIN {X 0,Y 446.428,Z 61.878,A -85,B 0,C 180,E1 -8760.249,E2 -8760.249} C_VEL
LIN {X 0,Y 446.445,Z 61.872,A -85,B 0,C 180,E1 -8763.453,E2 -8763.453} C_VEL
LIN {X 0,Y 446.408,Z 61.874,A -85,B 0,C 180,E1 -8766.744,E2 -8766.744} C_VEL
LIN {X 0,Y 446.478,Z 61.871,A -85,B 0,C 180,E1 -8769.528,E2 -8769.528} C_VEL
LIN {X 0,Y 446.429,Z 61.872,A -85,B 0,C 180,E1 -8772.604,E2 -8772.604} C_VEL
LIN {X 0,Y 446.451,Z 61.872,A -85,B 0,C 180,E1 -8775.104,E2 -8775.104} C_VEL
LIN {X 0,Y 446.427,Z 61.872,A -85,B 0,C 180,E1 -8778.609,E2 -8778.609} C_VEL
LIN {X 0,Y 446.441,Z 61.874,A -85,B 0,C 180,E1 -8780.973,E2 -8780.973} C_VEL
LIN {X 0,Y 446.419,Z 61.873,A -85,B 0,C 180,E1 -8784.374,E2 -8784.374} C_VEL
LIN {X 0,Y 446.422,Z 61.874,A -85,B 0,C 180,E1 -8787.638,E2 -8787.638} C_VEL
LIN {X 0,Y 446.448,Z 61.874,A -85,B 0,C 180,E1 -8790.791,E2 -8790.791} C_VEL
LIN {X 0,Y 446.477,Z 61.866,A -85,B 0,C 180,E1 -8793.848,E2 -8793.848} C_VEL
LIN {X 0,Y 446.428,Z 61.88,A -85,B 0,C 180,E1 -8796.823,E2 -8796.823} C_VEL
LIN {X 0,Y 446.443,Z 61.87,A -85,B 0,C 180,E1 -8799.737,E2 -8799.737} C_VEL
LIN {X 0,Y 446.456,Z 61.876,A -85,B 0,C 180,E1 -8802.597,E2 -8802.597} C_VEL
LIN {X 0,Y 446.468,Z 61.867,A -85,B 0,C 180,E1 -8805.412,E2 -8805.412} C_VEL
LIN {X 0,Y 446.516,Z 61.865,A -85,B 0,C 180,E1 -8808.193,E2 -8808.193} C_VEL
LIN {X 0,Y 446.6,Z 61.852,A -85,B 0,C 180,E1 -8811.858,E2 -8811.858} C_VEL
LIN {X 0,Y 446.642,Z 61.849,A -85,B 0,C 180,E1 -8814.583,E2 -8814.583} C_VEL
LIN {X 0,Y 446.661,Z 61.85,A -85,B 0,C 180,E1 -8818.197,E2 -8818.197} C_VEL
LIN {X 0,Y 446.791,Z 61.833,A -85,B 0,C 180,E1 -8820,E2 -8820} C_VEL
LIN {X 0,Y 446.683,Z 61.841,A -85,B 0,C 180,E1 -8822.706,E2 -8822.706} C_VEL
LIN {X 0,Y 446.619,Z 61.851,A -85,B 0,C 180,E1 -8826.324,E2 -8826.324} C_VEL
LIN {X 0,Y 446.521,Z 61.865,A -85,B 0,C 180,E1 -8829.97,E2 -8829.97} C_VEL
LIN {X 0,Y 446.521,Z 61.86,A -85,B 0,C 180,E1 -8832.73,E2 -8832.73} C_VEL
LIN {X 0,Y 446.488,Z 61.864,A -85,B 0,C 180,E1 -8836.459,E2 -8836.459} C_VEL
LIN {X 0,Y 446.468,Z 61.872,A -85,B 0,C 180,E1 -8839.304,E2 -8839.304} C_VEL
LIN {X 0,Y 446.418,Z 61.873,A -85,B 0,C 180,E1 -8842.2,E2 -8842.2} C_VEL
LIN {X 0,Y 446.437,Z 61.876,A -85,B 0,C 180,E1 -8845.154,E2 -8845.154} C_VEL
LIN {X 0,Y 446.485,Z 61.865,A -85,B 0,C 180,E1 -8848.179,E2 -8848.179} C_VEL
LIN {X 0,Y 446.419,Z 61.874,A -85,B 0,C 180,E1 -8851.775,E2 -8851.775} C_VEL
LIN {X 0,Y 446.424,Z 61.874,A -85,B 0,C 180,E1 -8854.524,E2 -8854.524} C_VEL
LIN {X 0,Y 446.413,Z 61.874,A -85,B 0,C 180,E1 -8858.079,E2 -8858.079} C_VEL
LIN {X 0,Y 446.406,Z 61.876,A -85,B 0,C 180,E1 -8861.394,E2 -8861.394} C_VEL
LIN {X 0,Y 446.451,Z 61.871,A -85,B 0,C 180,E1 -8865.104,E2 -8865.104} C_VEL
LIN {X 0,Y 446.42,Z 61.88,A -85,B 0,C 180,E1 -8868.608,E2 -8868.608} C_VEL
LIN {X 0,Y 446.412,Z 61.875,A -85,B 0,C 180,E1 -8871.922,E2 -8871.922} C_VEL
LIN {X 0,Y 446.43,Z 61.872,A -85,B 0,C 180,E1 -8875.477,E2 -8875.477} C_VEL
LIN {X 0,Y 446.418,Z 61.875,A -85,B 0,C 180,E1 -8878.7,E2 -8878.7} C_VEL
LIN {X 0,Y 446.453,Z 61.872,A -85,B 0,C 180,E1 -8881.83,E2 -8881.83} C_VEL
LIN {X 0,Y 446.424,Z 61.873,A -85,B 0,C 180,E1 -8884.846,E2 -8884.846} C_VEL
LIN {X 0,Y 446.452,Z 61.873,A -85,B 0,C 180,E1 -8888.246,E2 -8888.246} C_VEL
LIN {X 0,Y 446.453,Z 61.874,A -85,B 0,C 180,E1 -8891.649,E2 -8891.649} C_VEL
LIN {X 0,Y 446.51,Z 61.867,A -85,B 0,C 180,E1 -8894.48,E2 -8894.48} C_VEL
LIN {X 0,Y 446.5,Z 61.896,A -85,B 0,C 180,E1 -8896.344,E2 -8896.344} C_VEL
LIN {X 0,Y 447.702,Z 70.033,A -85,B 0,C 180,E1 -8898.225,E2 -8898.225} C_VEL
LIN {X 0,Y 447.6,Z 75.668,A -85,B 0,C 180,E1 -8899.464,E2 -8899.464} C_VEL
LIN {X 0,Y 450.66,Z 91.746,A -85,B 0,C 180,E1 -8899.837,E2 -8899.837} C_VEL
LIN {X 0,Y 450.422,Z 119.132,A -85,B 0,C 180,E1 -8900.273,E2 -8900.273} C_VEL
LIN {X 0,Y 449.636,Z 124.977,A -85,B 0,C 180,E1 -8900.341,E2 -8900.341} C_VEL
LIN {X 0,Y 443.899,Z 143.957,A -85,B 0,C 180,E1 -8900.454,E2 -8900.454} C_VEL
LIN {X 0,Y 443.238,Z 149.797,A -85,B 0,C 180,E1 -8900.527,E2 -8900.527} C_VEL
LIN {X 0,Y 442.861,Z 183.56,A -85,B 0,C 180,E1 -8901.099,E2 -8901.099} C_VEL
LIN {X 0,Y 442.632,Z 197.138,A -85,B 0,C 180,E1 -8901.526,E2 -8901.526} C_VEL
LIN {X 0,Y 442.201,Z 209.904,A -85,B 0,C 180,E1 -8902.121,E2 -8902.121} C_VEL
LIN {X 0,Y 441.833,Z 222.299,A -85,B 0,C 180,E1 -8902.919,E2 -8902.919} C_VEL
LIN {X 0,Y 441.181,Z 233.4,A -85,B 0,C 180,E1 -8903.827,E2 -8903.827} C_VEL
LIN {X 0,Y 440.7,Z 242.371,A -85,B 0,C 180,E1 -8904.739,E2 -8904.739} C_VEL
LIN {X 0,Y 440.177,Z 251.601,A -85,B 0,C 180,E1 -8905.88,E2 -8905.88} C_VEL
LIN {X 0,Y 439.574,Z 260.54,A -85,B 0,C 180,E1 -8907.251,E2 -8907.251} C_VEL
LIN {X 0,Y 439.195,Z 267.743,A -85,B 0,C 180,E1 -8908.625,E2 -8908.625} C_VEL
LIN {X 0,Y 438.794,Z 273.531,A -85,B 0,C 180,E1 -8910,E2 -8910} C_VEL
LIN {X 0,Y 438.574,Z 278.09,A -85,B 0,C 180,E1 -8911.378,E2 -8911.378} C_VEL
LIN {X 0,Y 438.513,Z 281.56,A -85,B 0,C 180,E1 -8912.756,E2 -8912.756} C_VEL
LIN {X 0,Y 438.446,Z 283.321,A -85,B 0,C 180,E1 -8913.676,E2 -8913.676} C_VEL
LIN {X 0,Y 438.398,Z 285.598,A -85,B 0,C 180,E1 -8915.52,E2 -8915.52} C_VEL
LIN {X 0,Y 438.431,Z 286.157,A -85,B 0,C 180,E1 -8916.443,E2 -8916.443} C_VEL
LIN {X 0,Y 438.359,Z 286.295,A -85,B 0,C 180,E1 -8917.369,E2 -8917.369} C_VEL
LIN {X 0,Y 438.332,Z 285.384,A -85,B 0,C 180,E1 -8919.227,E2 -8919.227} C_VEL
LIN {X 0,Y 438.363,Z 284.344,A -85,B 0,C 180,E1 -8920.158,E2 -8920.158} C_VEL
LIN {X 0,Y 438.492,Z 282.846,A -85,B 0,C 180,E1 -8921.089,E2 -8921.089} C_VEL
LIN {X 0,Y 438.676,Z 280.435,A -85,B 0,C 180,E1 -8922.235,E2 -8922.235} C_VEL
LIN {X 0,Y 438.934,Z 275.677,A -85,B 0,C 180,E1 -8923.897,E2 -8923.897} C_VEL
LIN {X 0,Y 439.399,Z 269.329,A -85,B 0,C 180,E1 -8925.54,E2 -8925.54} C_VEL
LIN {X 0,Y 439.86,Z 262.376,A -85,B 0,C 180,E1 -8926.954,E2 -8926.954} C_VEL
LIN {X 0,Y 440.487,Z 253.596,A -85,B 0,C 180,E1 -8928.368,E2 -8928.368} C_VEL
LIN {X 0,Y 441.139,Z 244.55,A -85,B 0,C 180,E1 -8929.546,E2 -8929.546} C_VEL
LIN {X 0,Y 441.732,Z 234.542,A -85,B 0,C 180,E1 -8930.611,E2 -8930.611} C_VEL
LIN {X 0,Y 442.372,Z 223.362,A -85,B 0,C 180,E1 -8931.555,E2 -8931.555} C_VEL
LIN {X 0,Y 443.089,Z 210.766,A -85,B 0,C 180,E1 -8932.376,E2 -8932.376} C_VEL
LIN {X 0,Y 443.593,Z 198.018,A -85,B 0,C 180,E1 -8932.989,E2 -8932.989} C_VEL
LIN {X 0,Y 443.961,Z 185.122,A -85,B 0,C 180,E1 -8933.406,E2 -8933.406} C_VEL
LIN {X 0,Y 444.189,Z 163.877,A -85,B 0,C 180,E1 -8933.795,E2 -8933.795} C_VEL
LIN {X 0,Y 444.88,Z 92.209,A -85,B 0,C 180,E1 -8934.97,E2 -8934.97} C_VEL
LIN {X 0,Y 441.145,Z 76.095,A -85,B 0,C 180,E1 -8935.449,E2 -8935.449} C_VEL
LIN {X 0,Y 441.09,Z 71.556,A -85,B 0,C 180,E1 -8936.496,E2 -8936.496} C_VEL
LIN {X 0,Y 439.437,Z 62.75,A -85,B 0,C 180,E1 -8938.672,E2 -8938.672} C_VEL
LIN {X 0,Y 439.348,Z 62.761,A -85,B 0,C 180,E1 -8942.025,E2 -8942.025} C_VEL
LIN {X 0,Y 439.386,Z 62.752,A -85,B 0,C 180,E1 -8945.338,E2 -8945.338} C_VEL
LIN {X 0,Y 439.353,Z 62.757,A -85,B 0,C 180,E1 -8948.599,E2 -8948.599} C_VEL
LIN {X 0,Y 439.362,Z 62.755,A -85,B 0,C 180,E1 -8951.252,E2 -8951.252} C_VEL
LIN {X 0,Y 439.375,Z 62.742,A -85,B 0,C 180,E1 -8954.733,E2 -8954.733} C_VEL
LIN {X 0,Y 439.348,Z 62.758,A -85,B 0,C 180,E1 -8957.789,E2 -8957.789} C_VEL
LIN {X 0,Y 439.349,Z 62.758,A -85,B 0,C 180,E1 -8961.401,E2 -8961.401} C_VEL
LIN {X 0,Y 439.389,Z 62.748,A -85,B 0,C 180,E1 -8964.843,E2 -8964.843} C_VEL
LIN {X 0,Y 439.348,Z 62.751,A -85,B 0,C 180,E1 -8968.137,E2 -8968.137} C_VEL
LIN {X 0,Y 439.38,Z 62.753,A -85,B 0,C 180,E1 -8971.323,E2 -8971.323} C_VEL
LIN {X 0,Y 439.356,Z 62.754,A -85,B 0,C 180,E1 -8974.412,E2 -8974.412} C_VEL
LIN {X 0,Y 439.365,Z 62.751,A -85,B 0,C 180,E1 -8977.424,E2 -8977.424} C_VEL
LIN {X 0,Y 439.444,Z 62.748,A -85,B 0,C 180,E1 -8980.663,E2 -8980.663} C_VEL
LIN {X 0,Y 439.448,Z 62.742,A -85,B 0,C 180,E1 -8984.224,E2 -8984.224} C_VEL
LIN {X 0,Y 439.486,Z 62.732,A -85,B 0,C 180,E1 -8988.001,E2 -8988.001} C_VEL
LIN {X 0,Y 439.505,Z 62.735,A -85,B 0,C 180,E1 -8991.725,E2 -8991.725} C_VEL
LIN {X 0,Y 439.595,Z 62.723,A -85,B 0,C 180,E1 -8994.495,E2 -8994.495} C_VEL
LIN {X 0,Y 439.633,Z 62.723,A -85,B 0,C 180,E1 -8998.168,E2 -8998.168} C_VEL
LIN {X 0,Y 439.588,Z 62.722,A -85,B 0,C 180,E1 -9000.916,E2 -9000.916} C_VEL
LIN {X 0,Y 439.608,Z 62.723,A -85,B 0,C 180,E1 -9002.749,E2 -9002.749} C_VEL
LIN {X 0,Y 439.562,Z 62.726,A -85,B 0,C 180,E1 -9006.426,E2 -9006.426} C_VEL
LIN {X 0,Y 439.494,Z 62.737,A -85,B 0,C 180,E1 -9009.202,E2 -9009.202} C_VEL
LIN {X 0,Y 439.468,Z 62.736,A -85,B 0,C 180,E1 -9012.937,E2 -9012.937} C_VEL
LIN {X 0,Y 439.447,Z 62.737,A -85,B 0,C 180,E1 -9016.347,E2 -9016.347} C_VEL
LIN {X 0,Y 439.404,Z 62.753,A -85,B 0,C 180,E1 -9019.626,E2 -9019.626} C_VEL
LIN {X 0,Y 439.366,Z 62.747,A -85,B 0,C 180,E1 -9022.575,E2 -9022.575} C_VEL
LIN {X 0,Y 439.388,Z 62.75,A -85,B 0,C 180,E1 -9025.586,E2 -9025.586} C_VEL
LIN {X 0,Y 439.42,Z 62.747,A -85,B 0,C 180,E1 -9028.673,E2 -9028.673} C_VEL
LIN {X 0,Y 439.372,Z 62.751,A -85,B 0,C 180,E1 -9032.03,E2 -9032.03} C_VEL
LIN {X 0,Y 439.397,Z 62.74,A -85,B 0,C 180,E1 -9035.34,E2 -9035.34} C_VEL
LIN {X 0,Y 439.38,Z 62.751,A -85,B 0,C 180,E1 -9038.595,E2 -9038.595} C_VEL
LIN {X 0,Y 439.391,Z 62.751,A -85,B 0,C 180,E1 -9041.257,E2 -9041.257} C_VEL
LIN {X 0,Y 439.402,Z 62.753,A -85,B 0,C 180,E1 -9044.729,E2 -9044.729} C_VEL
LIN {X 0,Y 439.398,Z 62.748,A -85,B 0,C 180,E1 -9047.796,E2 -9047.796} C_VEL
LIN {X 0,Y 439.439,Z 62.746,A -85,B 0,C 180,E1 -9050.228,E2 -9050.228} C_VEL
LIN {X 0,Y 439.376,Z 62.754,A -85,B 0,C 180,E1 -9053.713,E2 -9053.713} C_VEL
LIN {X 0,Y 439.375,Z 62.757,A -85,B 0,C 180,E1 -9057.054,E2 -9057.054} C_VEL
LIN {X 0,Y 439.385,Z 62.759,A -85,B 0,C 180,E1 -9060.274,E2 -9060.274} C_VEL
LIN {X 0,Y 439.493,Z 62.928,A -85,B 0,C 180,E1 -9062.194,E2 -9062.194} C_VEL
LIN {X 0,Y 442.276,Z 76.197,A -85,B 0,C 180,E1 -9064.926,E2 -9064.926} C_VEL
LIN {X 0,Y 442.513,Z 79.74,A -85,B 0,C 180,E1 -9065.61,E2 -9065.61} C_VEL
LIN {X 0,Y 441.484,Z 95.603,A -85,B 0,C 180,E1 -9068.522,E2 -9068.522} C_VEL
LIN {X 0,Y 440.576,Z 112.521,A -85,B 0,C 180,E1 -9071.588,E2 -9071.588} C_VEL
LIN {X 0,Y 444.179,Z 134.532,A -85,B 0,C 180,E1 -9072.13,E2 -9072.13} C_VEL
LIN {X 0,Y 444.497,Z 140.485,A -85,B 0,C 180,E1 -9072.245,E2 -9072.245} C_VEL
LIN {X 0,Y 443.696,Z 221.053,A -85,B 0,C 180,E1 -9073.582,E2 -9073.582} C_VEL
LIN {X 0,Y 443.192,Z 234.317,A -85,B 0,C 180,E1 -9073.977,E2 -9073.977} C_VEL
LIN {X 0,Y 442.523,Z 247.595,A -85,B 0,C 180,E1 -9074.572,E2 -9074.572} C_VEL
LIN {X 0,Y 441.883,Z 258.756,A -85,B 0,C 180,E1 -9075.257,E2 -9075.257} C_VEL
LIN {X 0,Y 441.129,Z 270.353,A -85,B 0,C 180,E1 -9076.173,E2 -9076.173} C_VEL
LIN {X 0,Y 440.459,Z 280.806,A -85,B 0,C 180,E1 -9077.209,E2 -9077.209} C_VEL
LIN {X 0,Y 439.921,Z 289.368,A -85,B 0,C 180,E1 -9078.247,E2 -9078.247} C_VEL
LIN {X 0,Y 439.304,Z 297.28,A -85,B 0,C 180,E1 -9079.398,E2 -9079.398} C_VEL
LIN {X 0,Y 438.892,Z 305.036,A -85,B 0,C 180,E1 -9080.785,E2 -9080.785} C_VEL
LIN {X 0,Y 438.587,Z 311.271,A -85,B 0,C 180,E1 -9082.171,E2 -9082.171} C_VEL
LIN {X 0,Y 438.413,Z 316.583,A -85,B 0,C 180,E1 -9083.666,E2 -9083.666} C_VEL
LIN {X 0,Y 438.338,Z 321.163,A -85,B 0,C 180,E1 -9085.402,E2 -9085.402} C_VEL
LIN {X 0,Y 438.29,Z 322.917,A -85,B 0,C 180,E1 -9086.322,E2 -9086.322} C_VEL
LIN {X 0,Y 438.375,Z 324.262,A -85,B 0,C 180,E1 -9087.243,E2 -9087.243} C_VEL
LIN {X 0,Y 438.313,Z 325.759,A -85,B 0,C 180,E1 -9089.081,E2 -9089.081} C_VEL
LIN {X 0,Y 438.32,Z 325.878,A -85,B 0,C 180,E1 -9090,E2 -9090} C_VEL
LIN {X 0,Y 438.321,Z 324.937,A -85,B 0,C 180,E1 -9091.837,E2 -9091.837} C_VEL
LIN {X 0,Y 438.381,Z 323.882,A -85,B 0,C 180,E1 -9092.756,E2 -9092.756} C_VEL
LIN {X 0,Y 438.32,Z 322.365,A -85,B 0,C 180,E1 -9093.677,E2 -9093.677} C_VEL
LIN {X 0,Y 438.396,Z 319.3,A -85,B 0,C 180,E1 -9095.058,E2 -9095.058} C_VEL
LIN {X 0,Y 438.367,Z 315.159,A -85,B 0,C 180,E1 -9096.443,E2 -9096.443} C_VEL
LIN {X 0,Y 438.609,Z 308.823,A -85,B 0,C 180,E1 -9098.059,E2 -9098.059} C_VEL
LIN {X 0,Y 438.873,Z 301.914,A -85,B 0,C 180,E1 -9099.447,E2 -9099.447} C_VEL
LIN {X 0,Y 439.192,Z 294.859,A -85,B 0,C 180,E1 -9100.604,E2 -9100.604} C_VEL
LIN {X 0,Y 439.744,Z 286.368,A -85,B 0,C 180,E1 -9101.757,E2 -9101.757} C_VEL
LIN {X 0,Y 440.255,Z 277.047,A -85,B 0,C 180,E1 -9102.796,E2 -9102.796} C_VEL
LIN {X 0,Y 440.835,Z 265.457,A -85,B 0,C 180,E1 -9103.835,E2 -9103.835} C_VEL
LIN {X 0,Y 441.465,Z 254.063,A -85,B 0,C 180,E1 -9104.639,E2 -9104.639} C_VEL
LIN {X 0,Y 442.024,Z 242.412,A -85,B 0,C 180,E1 -9105.268,E2 -9105.268} C_VEL
LIN {X 0,Y 442.483,Z 230.82,A -85,B 0,C 180,E1 -9105.724,E2 -9105.724} C_VEL
LIN {X 0,Y 442.813,Z 217.294,A -85,B 0,C 180,E1 -9106.066,E2 -9106.066} C_VEL
LIN {X 0,Y 443.407,Z 136.171,A -85,B 0,C 180,E1 -9107.384,E2 -9107.384} C_VEL
LIN {X 0,Y 440.164,Z 112.687,A -85,B 0,C 180,E1 -9107.9,E2 -9107.9} C_VEL
LIN {X 0,Y 440.863,Z 96.484,A -85,B 0,C 180,E1 -9110.775,E2 -9110.775} C_VEL
LIN {X 0,Y 441.907,Z 77.486,A -85,B 0,C 180,E1 -9114.175,E2 -9114.175} C_VEL
LIN {X 0,Y 441.361,Z 72.523,A -85,B 0,C 180,E1 -9115.111,E2 -9115.111} C_VEL
LIN {X 0,Y 439.498,Z 62.739,A -85,B 0,C 180,E1 -9117.048,E2 -9117.048} C_VEL
LIN {X 0,Y 439.381,Z 62.756,A -85,B 0,C 180,E1 -9120.261,E2 -9120.261} C_VEL
LIN {X 0,Y 439.397,Z 62.753,A -85,B 0,C 180,E1 -9123.724,E2 -9123.724} C_VEL
LIN {X 0,Y 439.356,Z 62.753,A -85,B 0,C 180,E1 -9126.888,E2 -9126.888} C_VEL
LIN {X 0,Y 439.413,Z 62.751,A -85,B 0,C 180,E1 -9129.851,E2 -9129.851} C_VEL
LIN {X 0,Y 439.381,Z 62.75,A -85,B 0,C 180,E1 -9132.627,E2 -9132.627} C_VEL
LIN {X 0,Y 439.399,Z 62.752,A -85,B 0,C 180,E1 -9135.27,E2 -9135.27} C_VEL
LIN {X 0,Y 439.388,Z 62.75,A -85,B 0,C 180,E1 -9138.743,E2 -9138.743} C_VEL
LIN {X 0,Y 439.372,Z 62.754,A -85,B 0,C 180,E1 -9141.608,E2 -9141.608} C_VEL
LIN {X 0,Y 439.399,Z 62.751,A -85,B 0,C 180,E1 -9144.844,E2 -9144.844} C_VEL
LIN {X 0,Y 439.372,Z 62.751,A -85,B 0,C 180,E1 -9148.14,E2 -9148.14} C_VEL
LIN {X 0,Y 439.432,Z 62.745,A -85,B 0,C 180,E1 -9151.598,E2 -9151.598} C_VEL
LIN {X 0,Y 439.404,Z 62.749,A -85,B 0,C 180,E1 -9154.415,E2 -9154.415} C_VEL
LIN {X 0,Y 439.364,Z 62.753,A -85,B 0,C 180,E1 -9157.425,E2 -9157.425} C_VEL
LIN {X 0,Y 439.44,Z 62.75,A -85,B 0,C 180,E1 -9160.663,E2 -9160.663} C_VEL
LIN {X 0,Y 439.461,Z 62.743,A -85,B 0,C 180,E1 -9164.225,E2 -9164.225} C_VEL
LIN {X 0,Y 439.483,Z 62.739,A -85,B 0,C 180,E1 -9168.001,E2 -9168.001} C_VEL
LIN {X 0,Y 439.547,Z 62.73,A -85,B 0,C 180,E1 -9171.726,E2 -9171.726} C_VEL
LIN {X 0,Y 439.617,Z 62.725,A -85,B 0,C 180,E1 -9174.496,E2 -9174.496} C_VEL
LIN {X 0,Y 439.631,Z 62.726,A -85,B 0,C 180,E1 -9178.168,E2 -9178.168} C_VEL
LIN {X 0,Y 439.76,Z 62.709,A -85,B 0,C 180,E1 -9180,E2 -9180} C_VEL
LIN {X 0,Y 439.633,Z 62.719,A -85,B 0,C 180,E1 -9182.749,E2 -9182.749} C_VEL
LIN {X 0,Y 439.591,Z 62.725,A -85,B 0,C 180,E1 -9186.426,E2 -9186.426} C_VEL
LIN {X 0,Y 439.495,Z 62.737,A -85,B 0,C 180,E1 -9189.202,E2 -9189.202} C_VEL
LIN {X 0,Y 439.465,Z 62.74,A -85,B 0,C 180,E1 -9192.938,E2 -9192.938} C_VEL
LIN {X 0,Y 439.446,Z 62.742,A -85,B 0,C 180,E1 -9196.348,E2 -9196.348} C_VEL
LIN {X 0,Y 439.402,Z 62.753,A -85,B 0,C 180,E1 -9199.627,E2 -9199.627} C_VEL
LIN {X 0,Y 439.363,Z 62.752,A -85,B 0,C 180,E1 -9202.576,E2 -9202.576} C_VEL
LIN {X 0,Y 439.386,Z 62.753,A -85,B 0,C 180,E1 -9205.586,E2 -9205.586} C_VEL
LIN {X 0,Y 439.417,Z 62.747,A -85,B 0,C 180,E1 -9208.674,E2 -9208.674} C_VEL
LIN {X 0,Y 439.369,Z 62.751,A -85,B 0,C 180,E1 -9212.03,E2 -9212.03} C_VEL
LIN {X 0,Y 439.393,Z 62.751,A -85,B 0,C 180,E1 -9215.34,E2 -9215.34} C_VEL
LIN {X 0,Y 439.369,Z 62.755,A -85,B 0,C 180,E1 -9218.597,E2 -9218.597} C_VEL
LIN {X 0,Y 439.368,Z 62.754,A -85,B 0,C 180,E1 -9221.254,E2 -9221.254} C_VEL
LIN {X 0,Y 439.399,Z 62.754,A -85,B 0,C 180,E1 -9224.73,E2 -9224.73} C_VEL
LIN {X 0,Y 439.386,Z 62.749,A -85,B 0,C 180,E1 -9227.795,E2 -9227.795} C_VEL
LIN {X 0,Y 439.36,Z 62.756,A -85,B 0,C 180,E1 -9230.22,E2 -9230.22} C_VEL
LIN {X 0,Y 439.373,Z 62.751,A -85,B 0,C 180,E1 -9233.713,E2 -9233.713} C_VEL
LIN {X 0,Y 439.375,Z 62.751,A -85,B 0,C 180,E1 -9237.054,E2 -9237.054} C_VEL
LIN {X 0,Y 439.38,Z 62.756,A -85,B 0,C 180,E1 -9240.274,E2 -9240.274} C_VEL
LIN {X 0,Y 439.382,Z 62.75,A -85,B 0,C 180,E1 -9243.393,E2 -9243.393} C_VEL
LIN {X 0,Y 439.384,Z 62.752,A -85,B 0,C 180,E1 -9246.43,E2 -9246.43} C_VEL
LIN {X 0,Y 439.391,Z 62.75,A -85,B 0,C 180,E1 -9249.397,E2 -9249.397} C_VEL
LIN {X 0,Y 439.426,Z 62.75,A -85,B 0,C 180,E1 -9252.31,E2 -9252.31} C_VEL
LIN {X 0,Y 439.449,Z 62.748,A -85,B 0,C 180,E1 -9255.174,E2 -9255.174} C_VEL
LIN {X 0,Y 439.481,Z 62.798,A -85,B 0,C 180,E1 -9256.186,E2 -9256.186} C_VEL
LIN {X 0,Y 440.689,Z 70.693,A -85,B 0,C 180,E1 -9258.035,E2 -9258.035} C_VEL
LIN {X 0,Y 440.665,Z 76.13,A -85,B 0,C 180,E1 -9259.216,E2 -9259.216} C_VEL
LIN {X 0,Y 443.808,Z 92.324,A -85,B 0,C 180,E1 -9259.601,E2 -9259.601} C_VEL
LIN {X 0,Y 443.238,Z 149.797,A -85,B 0,C 180,E1 -9260.527,E2 -9260.527} C_VEL
LIN {X 0,Y 442.562,Z 155.641,A -85,B 0,C 180,E1 -9260.599,E2 -9260.599} C_VEL
LIN {X 0,Y 436.789,Z 174.608,A -85,B 0,C 180,E1 -9260.715,E2 -9260.715} C_VEL
LIN {X 0,Y 436.089,Z 180.436,A -85,B 0,C 180,E1 -9260.802,E2 -9260.802} C_VEL
LIN {X 0,Y 435.857,Z 193.526,A -85,B 0,C 180,E1 -9261.16,E2 -9261.16} C_VEL
LIN {X 0,Y 435.455,Z 206.285,A -85,B 0,C 180,E1 -9261.707,E2 -9261.707} C_VEL
LIN {X 0,Y 435.042,Z 218.936,A -85,B 0,C 180,E1 -9262.458,E2 -9262.458} C_VEL
LIN {X 0,Y 434.501,Z 229.485,A -85,B 0,C 180,E1 -9263.266,E2 -9263.266} C_VEL
LIN {X 0,Y 433.884,Z 240.266,A -85,B 0,C 180,E1 -9264.306,E2 -9264.306} C_VEL
LIN {X 0,Y 433.358,Z 249.061,A -85,B 0,C 180,E1 -9265.349,E2 -9265.349} C_VEL
LIN {X 0,Y 432.74,Z 258.62,A -85,B 0,C 180,E1 -9266.742,E2 -9266.742} C_VEL
LIN {X 0,Y 432.224,Z 266.25,A -85,B 0,C 180,E1 -9268.137,E2 -9268.137} C_VEL
LIN {X 0,Y 431.882,Z 272.372,A -85,B 0,C 180,E1 -9269.534,E2 -9269.534} C_VEL
LIN {X 0,Y 431.529,Z 277.252,A -85,B 0,C 180,E1 -9270.933,E2 -9270.933} C_VEL
LIN {X 0,Y 431.489,Z 281.009,A -85,B 0,C 180,E1 -9272.334,E2 -9272.334} C_VEL
LIN {X 0,Y 431.344,Z 283.771,A -85,B 0,C 180,E1 -9273.737,E2 -9273.737} C_VEL
LIN {X 0,Y 431.323,Z 285.989,A -85,B 0,C 180,E1 -9275.611,E2 -9275.611} C_VEL
LIN {X 0,Y 431.333,Z 286.508,A -85,B 0,C 180,E1 -9276.549,E2 -9276.549} C_VEL
LIN {X 0,Y 431.265,Z 286.31,A -85,B 0,C 180,E1 -9278.434,E2 -9278.434} C_VEL
LIN {X 0,Y 431.261,Z 285.634,A -85,B 0,C 180,E1 -9279.379,E2 -9279.379} C_VEL
LIN {X 0,Y 431.309,Z 284.548,A -85,B 0,C 180,E1 -9280.326,E2 -9280.326} C_VEL
LIN {X 0,Y 431.43,Z 283.008,A -85,B 0,C 180,E1 -9281.273,E2 -9281.273} C_VEL
LIN {X 0,Y 431.656,Z 279.902,A -85,B 0,C 180,E1 -9282.697,E2 -9282.697} C_VEL
LIN {X 0,Y 431.926,Z 275.71,A -85,B 0,C 180,E1 -9284.127,E2 -9284.127} C_VEL
LIN {X 0,Y 432.411,Z 269.29,A -85,B 0,C 180,E1 -9285.798,E2 -9285.798} C_VEL
LIN {X 0,Y 432.923,Z 262.229,A -85,B 0,C 180,E1 -9287.234,E2 -9287.234} C_VEL
LIN {X 0,Y 433.607,Z 253.335,A -85,B 0,C 180,E1 -9288.67,E2 -9288.67} C_VEL
LIN {X 0,Y 434.313,Z 244.174,A -85,B 0,C 180,E1 -9289.866,E2 -9289.866} C_VEL
LIN {X 0,Y 434.983,Z 233.976,A -85,B 0,C 180,E1 -9290.945,E2 -9290.945} C_VEL
LIN {X 0,Y 435.655,Z 222.558,A -85,B 0,C 180,E1 -9291.904,E2 -9291.904} C_VEL
LIN {X 0,Y 436.371,Z 210.688,A -85,B 0,C 180,E1 -9292.677,E2 -9292.677} C_VEL
LIN {X 0,Y 436.874,Z 197.928,A -85,B 0,C 180,E1 -9293.292,E2 -9293.292} C_VEL
LIN {X 0,Y 437.303,Z 184.531,A -85,B 0,C 180,E1 -9293.721,E2 -9293.721} C_VEL
LIN {X 0,Y 437.616,Z 155.444,A -85,B 0,C 180,E1 -9294.238,E2 -9294.238} C_VEL
LIN {X 0,Y 438.241,Z 93.29,A -85,B 0,C 180,E1 -9295.274,E2 -9295.274} C_VEL
LIN {X 0,Y 434.269,Z 76.465,A -85,B 0,C 180,E1 -9295.776,E2 -9295.776} C_VEL
LIN {X 0,Y 433.891,Z 71.259,A -85,B 0,C 180,E1 -9297.016,E2 -9297.016} C_VEL
LIN {X 0,Y 432.366,Z 63.63,A -85,B 0,C 180,E1 -9298.948,E2 -9298.948} C_VEL
LIN {X 0,Y 432.312,Z 63.635,A -85,B 0,C 180,E1 -9302.289,E2 -9302.289} C_VEL
LIN {X 0,Y 432.34,Z 63.631,A -85,B 0,C 180,E1 -9305.63,E2 -9305.63} C_VEL
LIN {X 0,Y 432.318,Z 63.633,A -85,B 0,C 180,E1 -9308.71,E2 -9308.71} C_VEL
LIN {X 0,Y 432.304,Z 63.637,A -85,B 0,C 180,E1 -9311.801,E2 -9311.801} C_VEL
LIN {X 0,Y 432.335,Z 63.62,A -85,B 0,C 180,E1 -9314.348,E2 -9314.348} C_VEL
LIN {X 0,Y 432.304,Z 63.633,A -85,B 0,C 180,E1 -9317.019,E2 -9317.019} C_VEL
LIN {X 0,Y 432.29,Z 63.639,A -85,B 0,C 180,E1 -9319.828,E2 -9319.828} C_VEL
LIN {X 0,Y 432.295,Z 63.636,A -85,B 0,C 180,E1 -9323.02,E2 -9323.02} C_VEL
LIN {X 0,Y 432.333,Z 63.63,A -85,B 0,C 180,E1 -9326.002,E2 -9326.002} C_VEL
LIN {X 0,Y 432.334,Z 63.633,A -85,B 0,C 180,E1 -9329.494,E2 -9329.494} C_VEL
LIN {X 0,Y 432.315,Z 63.628,A -85,B 0,C 180,E1 -9331.872,E2 -9331.872} C_VEL
LIN {X 0,Y 432.351,Z 63.627,A -85,B 0,C 180,E1 -9335.547,E2 -9335.547} C_VEL
LIN {X 0,Y 432.353,Z 63.632,A -85,B 0,C 180,E1 -9339.046,E2 -9339.046} C_VEL
LIN {X 0,Y 432.361,Z 63.621,A -85,B 0,C 180,E1 -9342.01,E2 -9342.01} C_VEL
LIN {X 0,Y 432.384,Z 63.627,A -85,B 0,C 180,E1 -9344.926,E2 -9344.926} C_VEL
LIN {X 0,Y 432.462,Z 63.606,A -85,B 0,C 180,E1 -9347.803,E2 -9347.803} C_VEL
LIN {X 0,Y 432.465,Z 63.612,A -85,B 0,C 180,E1 -9351.59,E2 -9351.59} C_VEL
LIN {X 0,Y 432.55,Z 63.599,A -85,B 0,C 180,E1 -9354.405,E2 -9354.405} C_VEL
LIN {X 0,Y 432.602,Z 63.599,A -85,B 0,C 180,E1 -9358.138,E2 -9358.138} C_VEL
LIN {X 0,Y 432.549,Z 63.599,A -85,B 0,C 180,E1 -9360.931,E2 -9360.931} C_VEL
LIN {X 0,Y 432.562,Z 63.601,A -85,B 0,C 180,E1 -9362.794,E2 -9362.794} C_VEL
LIN {X 0,Y 432.575,Z 63.596,A -85,B 0,C 180,E1 -9365.594,E2 -9365.594} C_VEL
LIN {X 0,Y 432.465,Z 63.613,A -85,B 0,C 180,E1 -9368.41,E2 -9368.41} C_VEL
LIN {X 0,Y 432.462,Z 63.61,A -85,B 0,C 180,E1 -9372.196,E2 -9372.196} C_VEL
LIN {X 0,Y 432.428,Z 63.614,A -85,B 0,C 180,E1 -9376.039,E2 -9376.039} C_VEL
LIN {X 0,Y 432.389,Z 63.627,A -85,B 0,C 180,E1 -9379.485,E2 -9379.485} C_VEL
LIN {X 0,Y 432.319,Z 63.627,A -85,B 0,C 180,E1 -9382.964,E2 -9382.964} C_VEL
LIN {X 0,Y 432.352,Z 63.624,A -85,B 0,C 180,E1 -9386.033,E2 -9386.033} C_VEL
LIN {X 0,Y 432.345,Z 63.633,A -85,B 0,C 180,E1 -9389.187,E2 -9389.187} C_VEL
LIN {X 0,Y 432.326,Z 63.63,A -85,B 0,C 180,E1 -9392.443,E2 -9392.443} C_VEL
LIN {X 0,Y 432.347,Z 63.616,A -85,B 0,C 180,E1 -9395.632,E2 -9395.632} C_VEL
LIN {X 0,Y 432.343,Z 63.629,A -85,B 0,C 180,E1 -9398.714,E2 -9398.714} C_VEL
LIN {X 0,Y 432.336,Z 63.628,A -85,B 0,C 180,E1 -9401.797,E2 -9401.797} C_VEL
LIN {X 0,Y 432.336,Z 63.633,A -85,B 0,C 180,E1 -9404.347,E2 -9404.347} C_VEL
LIN {X 0,Y 432.323,Z 63.631,A -85,B 0,C 180,E1 -9407.015,E2 -9407.015} C_VEL
LIN {X 0,Y 432.344,Z 63.628,A -85,B 0,C 180,E1 -9409.819,E2 -9409.819} C_VEL
LIN {X 0,Y 432.309,Z 63.633,A -85,B 0,C 180,E1 -9413.022,E2 -9413.022} C_VEL
LIN {X 0,Y 432.362,Z 63.631,A -85,B 0,C 180,E1 -9415.996,E2 -9415.996} C_VEL
LIN {X 0,Y 432.35,Z 63.634,A -85,B 0,C 180,E1 -9419.489,E2 -9419.489} C_VEL
LIN {X 0,Y 432.435,Z 63.756,A -85,B 0,C 180,E1 -9421.88,E2 -9421.88} C_VEL
LIN {X 0,Y 435.097,Z 76.201,A -85,B 0,C 180,E1 -9424.502,E2 -9424.502} C_VEL
LIN {X 0,Y 435.641,Z 80.965,A -85,B 0,C 180,E1 -9425.454,E2 -9425.454} C_VEL
LIN {X 0,Y 434.447,Z 98.131,A -85,B 0,C 180,E1 -9428.655,E2 -9428.655} C_VEL
LIN {X 0,Y 433.675,Z 112.177,A -85,B 0,C 180,E1 -9431.245,E2 -9431.245} C_VEL
LIN {X 0,Y 437.384,Z 134.489,A -85,B 0,C 180,E1 -9431.812,E2 -9431.812} C_VEL
LIN {X 0,Y 437.855,Z 139.663,A -85,B 0,C 180,E1 -9431.923,E2 -9431.923} C_VEL
LIN {X 0,Y 436.973,Z 220.909,A -85,B 0,C 180,E1 -9433.292,E2 -9433.292} C_VEL
LIN {X 0,Y 436.401,Z 234.114,A -85,B 0,C 180,E1 -9433.69,E2 -9433.69} C_VEL
LIN {X 0,Y 435.766,Z 246.796,A -85,B 0,C 180,E1 -9434.267,E2 -9434.267} C_VEL
LIN {X 0,Y 435.026,Z 258.883,A -85,B 0,C 180,E1 -9435.019,E2 -9435.019} C_VEL
LIN {X 0,Y 434.239,Z 270.395,A -85,B 0,C 180,E1 -9435.95,E2 -9435.95} C_VEL
LIN {X 0,Y 433.491,Z 280.783,A -85,B 0,C 180,E1 -9437,E2 -9437} C_VEL
LIN {X 0,Y 432.941,Z 289.294,A -85,B 0,C 180,E1 -9438.055,E2 -9438.055} C_VEL
LIN {X 0,Y 432.205,Z 298.541,A -85,B 0,C 180,E1 -9439.459,E2 -9439.459} C_VEL
LIN {X 0,Y 431.771,Z 305.987,A -85,B 0,C 180,E1 -9440.868,E2 -9440.868} C_VEL
LIN {X 0,Y 431.45,Z 312.876,A -85,B 0,C 180,E1 -9442.512,E2 -9442.512} C_VEL
LIN {X 0,Y 431.336,Z 316.694,A -85,B 0,C 180,E1 -9443.673,E2 -9443.673} C_VEL
LIN {X 0,Y 431.265,Z 320.907,A -85,B 0,C 180,E1 -9445.326,E2 -9445.326} C_VEL
LIN {X 0,Y 431.282,Z 323.977,A -85,B 0,C 180,E1 -9447.198,E2 -9447.198} C_VEL
LIN {X 0,Y 431.243,Z 324.912,A -85,B 0,C 180,E1 -9448.132,E2 -9448.132} C_VEL
LIN {X 0,Y 431.226,Z 325.449,A -85,B 0,C 180,E1 -9449.066,E2 -9449.066} C_VEL
LIN {X 0,Y 431.231,Z 325.552,A -85,B 0,C 180,E1 -9450,E2 -9450} C_VEL
LIN {X 0,Y 431.243,Z 324.591,A -85,B 0,C 180,E1 -9451.868,E2 -9451.868} C_VEL
LIN {X 0,Y 431.308,Z 323.521,A -85,B 0,C 180,E1 -9452.802,E2 -9452.802} C_VEL
LIN {X 0,Y 431.222,Z 321.984,A -85,B 0,C 180,E1 -9453.738,E2 -9453.738} C_VEL
LIN {X 0,Y 431.298,Z 318.896,A -85,B 0,C 180,E1 -9455.142,E2 -9455.142} C_VEL
LIN {X 0,Y 431.289,Z 314.729,A -85,B 0,C 180,E1 -9456.55,E2 -9456.55} C_VEL
LIN {X 0,Y 431.555,Z 308.366,A -85,B 0,C 180,E1 -9458.192,E2 -9458.192} C_VEL
LIN {X 0,Y 431.837,Z 301.425,A -85,B 0,C 180,E1 -9459.602,E2 -9459.602} C_VEL
LIN {X 0,Y 432.176,Z 294.333,A -85,B 0,C 180,E1 -9460.778,E2 -9460.778} C_VEL
LIN {X 0,Y 432.729,Z 285.788,A -85,B 0,C 180,E1 -9461.951,E2 -9461.951} C_VEL
LIN {X 0,Y 433.339,Z 275.211,A -85,B 0,C 180,E1 -9463.124,E2 -9463.124} C_VEL
LIN {X 0,Y 433.961,Z 263.289,A -85,B 0,C 180,E1 -9464.179,E2 -9464.179} C_VEL
LIN {X 0,Y 434.656,Z 251.267,A -85,B 0,C 180,E1 -9464.993,E2 -9464.993} C_VEL
LIN {X 0,Y 435.242,Z 238.733,A -85,B 0,C 180,E1 -9465.632,E2 -9465.632} C_VEL
LIN {X 0,Y 435.75,Z 225.699,A -85,B 0,C 180,E1 -9466.093,E2 -9466.093} C_VEL
LIN {X 0,Y 436.011,Z 209.879,A -85,B 0,C 180,E1 -9466.414,E2 -9466.414} C_VEL
LIN {X 0,Y 436.5,Z 136.565,A -85,B 0,C 180,E1 -9467.621,E2 -9467.621} C_VEL
LIN {X 0,Y 433.162,Z 112.417,A -85,B 0,C 180,E1 -9468.153,E2 -9468.153} C_VEL
LIN {X 0,Y 433.878,Z 97.316,A -85,B 0,C 180,E1 -9470.876,E2 -9470.876} C_VEL
LIN {X 0,Y 434.955,Z 78.324,A -85,B 0,C 180,E1 -9474.332,E2 -9474.332} C_VEL
LIN {X 0,Y 434.152,Z 72.611,A -85,B 0,C 180,E1 -9475.437,E2 -9475.437} C_VEL
LIN {X 0,Y 432.454,Z 63.614,A -85,B 0,C 180,E1 -9477.263,E2 -9477.263} C_VEL
LIN {X 0,Y 432.348,Z 63.629,A -85,B 0,C 180,E1 -9480.51,E2 -9480.51} C_VEL
LIN {X 0,Y 432.359,Z 63.63,A -85,B 0,C 180,E1 -9484.003,E2 -9484.003} C_VEL
LIN {X 0,Y 432.331,Z 63.629,A -85,B 0,C 180,E1 -9487.198,E2 -9487.198} C_VEL
LIN {X 0,Y 432.341,Z 63.628,A -85,B 0,C 180,E1 -9490.18,E2 -9490.18} C_VEL
LIN {X 0,Y 432.317,Z 63.632,A -85,B 0,C 180,E1 -9493.061,E2 -9493.061} C_VEL
LIN {X 0,Y 432.332,Z 63.633,A -85,B 0,C 180,E1 -9495.665,E2 -9495.665} C_VEL
LIN {X 0,Y 432.332,Z 63.628,A -85,B 0,C 180,E1 -9498.398,E2 -9498.398} C_VEL
LIN {X 0,Y 432.335,Z 63.629,A -85,B 0,C 180,E1 -9501.85,E2 -9501.85} C_VEL
LIN {X 0,Y 432.339,Z 63.633,A -85,B 0,C 180,E1 -9505.323,E2 -9505.323} C_VEL
LIN {X 0,Y 432.321,Z 63.632,A -85,B 0,C 180,E1 -9508.654,E2 -9508.654} C_VEL
LIN {X 0,Y 432.381,Z 63.622,A -85,B 0,C 180,E1 -9511.877,E2 -9511.877} C_VEL
LIN {X 0,Y 432.351,Z 63.631,A -85,B 0,C 180,E1 -9514.999,E2 -9514.999} C_VEL
LIN {X 0,Y 432.357,Z 63.625,A -85,B 0,C 180,E1 -9518.046,E2 -9518.046} C_VEL
LIN {X 0,Y 432.384,Z 63.625,A -85,B 0,C 180,E1 -9521.03,E2 -9521.03} C_VEL
LIN {X 0,Y 432.429,Z 63.617,A -85,B 0,C 180,E1 -9523.961,E2 -9523.961} C_VEL
LIN {X 0,Y 432.458,Z 63.613,A -85,B 0,C 180,E1 -9527.804,E2 -9527.804} C_VEL
LIN {X 0,Y 432.491,Z 63.608,A -85,B 0,C 180,E1 -9531.59,E2 -9531.59} C_VEL
LIN {X 0,Y 432.594,Z 63.601,A -85,B 0,C 180,E1 -9534.406,E2 -9534.406} C_VEL
LIN {X 0,Y 432.601,Z 63.602,A -85,B 0,C 180,E1 -9538.138,E2 -9538.138} C_VEL
LIN {X 0,Y 432.73,Z 63.585,A -85,B 0,C 180,E1 -9540,E2 -9540} C_VEL
LIN {X 0,Y 432.585,Z 63.597,A -85,B 0,C 180,E1 -9542.794,E2 -9542.794} C_VEL
LIN {X 0,Y 432.585,Z 63.6,A -85,B 0,C 180,E1 -9545.594,E2 -9545.594} C_VEL
LIN {X 0,Y 432.463,Z 63.613,A -85,B 0,C 180,E1 -9548.41,E2 -9548.41} C_VEL
LIN {X 0,Y 432.459,Z 63.614,A -85,B 0,C 180,E1 -9552.197,E2 -9552.197} C_VEL
LIN {X 0,Y 432.43,Z 63.618,A -85,B 0,C 180,E1 -9556.039,E2 -9556.039} C_VEL
LIN {X 0,Y 432.386,Z 63.629,A -85,B 0,C 180,E1 -9559.485,E2 -9559.485} C_VEL
LIN {X 0,Y 432.317,Z 63.632,A -85,B 0,C 180,E1 -9562.965,E2 -9562.965} C_VEL
LIN {X 0,Y 432.35,Z 63.626,A -85,B 0,C 180,E1 -9566.034,E2 -9566.034} C_VEL
LIN {X 0,Y 432.343,Z 63.634,A -85,B 0,C 180,E1 -9569.188,E2 -9569.188} C_VEL
LIN {X 0,Y 432.323,Z 63.63,A -85,B 0,C 180,E1 -9572.443,E2 -9572.443} C_VEL
LIN {X 0,Y 432.344,Z 63.627,A -85,B 0,C 180,E1 -9575.632,E2 -9575.632} C_VEL
LIN {X 0,Y 432.331,Z 63.633,A -85,B 0,C 180,E1 -9578.713,E2 -9578.713} C_VEL
LIN {X 0,Y 432.309,Z 63.631,A -85,B 0,C 180,E1 -9581.801,E2 -9581.801} C_VEL
LIN {X 0,Y 432.334,Z 63.631,A -85,B 0,C 180,E1 -9584.348,E2 -9584.348} C_VEL
LIN {X 0,Y 432.318,Z 63.632,A -85,B 0,C 180,E1 -9587.017,E2 -9587.017} C_VEL
LIN {X 0,Y 432.315,Z 63.631,A -85,B 0,C 180,E1 -9589.824,E2 -9589.824} C_VEL
LIN {X 0,Y 432.306,Z 63.632,A -85,B 0,C 180,E1 -9593.022,E2 -9593.022} C_VEL
LIN {X 0,Y 432.361,Z 63.628,A -85,B 0,C 180,E1 -9595.997,E2 -9595.997} C_VEL
LIN {X 0,Y 432.349,Z 63.626,A -85,B 0,C 180,E1 -9599.49,E2 -9599.49} C_VEL
LIN {X 0,Y 432.349,Z 63.63,A -85,B 0,C 180,E1 -9601.875,E2 -9601.875} C_VEL
LIN {X 0,Y 432.365,Z 63.626,A -85,B 0,C 180,E1 -9605.544,E2 -9605.544} C_VEL
LIN {X 0,Y 432.353,Z 63.625,A -85,B 0,C 180,E1 -9609.046,E2 -9609.046} C_VEL
LIN {X 0,Y 432.374,Z 63.63,A -85,B 0,C 180,E1 -9612.011,E2 -9612.011} C_VEL
LIN {X 0,Y 432.397,Z 63.626,A -85,B 0,C 180,E1 -9614.927,E2 -9614.927} C_VEL
LIN {X 0,Y 432.45,Z 63.711,A -85,B 0,C 180,E1 -9616.023,E2 -9616.023} C_VEL
LIN {X 0,Y 433.747,Z 72.376,A -85,B 0,C 180,E1 -9618.078,E2 -9618.078} C_VEL
LIN {X 0,Y 433.69,Z 76.222,A -85,B 0,C 180,E1 -9618.945,E2 -9618.945} C_VEL
LIN {X 0,Y 436.984,Z 93.769,A -85,B 0,C 180,E1 -9619.373,E2 -9619.373} C_VEL
LIN {X 0,Y 436.089,Z 180.436,A -85,B 0,C 180,E1 -9620.802,E2 -9620.802} C_VEL
LIN {X 0,Y 435.396,Z 184.341,A -85,B 0,C 180,E1 -9620.863,E2 -9620.863} C_VEL
LIN {X 0,Y 432.525,Z 190.443,A -85,B 0,C 180,E1 -9620.932,E2 -9620.932} C_VEL
LIN {X 0,Y 429.578,Z 196.457,A -85,B 0,C 180,E1 -9621.049,E2 -9621.049} C_VEL
LIN {X 0,Y 428.764,Z 200.225,A -85,B 0,C 180,E1 -9621.186,E2 -9621.186} C_VEL
LIN {X 0,Y 428.333,Z 213.287,A -85,B 0,C 180,E1 -9621.865,E2 -9621.865} C_VEL
LIN {X 0,Y 427.879,Z 225.124,A -85,B 0,C 180,E1 -9622.687,E2 -9622.687} C_VEL
LIN {X 0,Y 427.214,Z 235.724,A -85,B 0,C 180,E1 -9623.625,E2 -9623.625} C_VEL
LIN {X 0,Y 426.551,Z 246.348,A -85,B 0,C 180,E1 -9624.801,E2 -9624.801} C_VEL
LIN {X 0,Y 425.998,Z 254.985,A -85,B 0,C 180,E1 -9625.98,E2 -9625.98} C_VEL
LIN {X 0,Y 425.432,Z 263.396,A -85,B 0,C 180,E1 -9627.396,E2 -9627.396} C_VEL
LIN {X 0,Y 424.974,Z 270.149,A -85,B 0,C 180,E1 -9628.816,E2 -9628.816} C_VEL
LIN {X 0,Y 424.546,Z 276.362,A -85,B 0,C 180,E1 -9630.475,E2 -9630.475} C_VEL
LIN {X 0,Y 424.434,Z 280.413,A -85,B 0,C 180,E1 -9631.898,E2 -9631.898} C_VEL
LIN {X 0,Y 424.354,Z 282.543,A -85,B 0,C 180,E1 -9632.848,E2 -9632.848} C_VEL
LIN {X 0,Y 424.204,Z 285.495,A -85,B 0,C 180,E1 -9634.752,E2 -9634.752} C_VEL
LIN {X 0,Y 424.267,Z 286.716,A -85,B 0,C 180,E1 -9636.326,E2 -9636.326} C_VEL
LIN {X 0,Y 424.182,Z 286.909,A -85,B 0,C 180,E1 -9637.617,E2 -9637.617} C_VEL
LIN {X 0,Y 424.174,Z 285.885,A -85,B 0,C 180,E1 -9639.537,E2 -9639.537} C_VEL
LIN {X 0,Y 424.262,Z 284.741,A -85,B 0,C 180,E1 -9640.499,E2 -9640.499} C_VEL
LIN {X 0,Y 424.564,Z 281.239,A -85,B 0,C 180,E1 -9642.403,E2 -9642.403} C_VEL
LIN {X 0,Y 424.813,Z 277.305,A -85,B 0,C 180,E1 -9643.88,E2 -9643.88} C_VEL
LIN {X 0,Y 425.209,Z 272.262,A -85,B 0,C 180,E1 -9645.335,E2 -9645.335} C_VEL
LIN {X 0,Y 425.756,Z 265.929,A -85,B 0,C 180,E1 -9646.78,E2 -9646.78} C_VEL
LIN {X 0,Y 426.326,Z 257.824,A -85,B 0,C 180,E1 -9648.253,E2 -9648.253} C_VEL
LIN {X 0,Y 427.051,Z 249.582,A -85,B 0,C 180,E1 -9649.467,E2 -9649.467} C_VEL
LIN {X 0,Y 427.781,Z 239.357,A -85,B 0,C 180,E1 -9650.697,E2 -9650.697} C_VEL
LIN {X 0,Y 428.569,Z 227.923,A -85,B 0,C 180,E1 -9651.779,E2 -9651.779} C_VEL
LIN {X 0,Y 429.286,Z 216.539,A -85,B 0,C 180,E1 -9652.627,E2 -9652.627} C_VEL
LIN {X 0,Y 429.905,Z 205.131,A -85,B 0,C 180,E1 -9653.281,E2 -9653.281} C_VEL
LIN {X 0,Y 430.343,Z 192.831,A -85,B 0,C 180,E1 -9653.793,E2 -9653.793} C_VEL
LIN {X 0,Y 430.656,Z 179.638,A -85,B 0,C 180,E1 -9654.143,E2 -9654.143} C_VEL
LIN {X 0,Y 431.687,Z 94.978,A -85,B 0,C 180,E1 -9655.574,E2 -9655.574} C_VEL
LIN {X 0,Y 427.394,Z 76.769,A -85,B 0,C 180,E1 -9656.132,E2 -9656.132} C_VEL
LIN {X 0,Y 426.704,Z 71.349,A -85,B 0,C 180,E1 -9657.463,E2 -9657.463} C_VEL
LIN {X 0,Y 425.3,Z 64.51,A -85,B 0,C 180,E1 -9659.254,E2 -9659.254} C_VEL
LIN {X 0,Y 425.27,Z 64.512,A -85,B 0,C 180,E1 -9662.559,E2 -9662.559} C_VEL
LIN {X 0,Y 425.293,Z 64.508,A -85,B 0,C 180,E1 -9665.337,E2 -9665.337} C_VEL
LIN {X 0,Y 425.276,Z 64.51,A -85,B 0,C 180,E1 -9668.901,E2 -9668.901} C_VEL
LIN {X 0,Y 425.257,Z 64.511,A -85,B 0,C 180,E1 -9672.656,E2 -9672.656} C_VEL
LIN {X 0,Y 425.286,Z 64.498,A -85,B 0,C 180,E1 -9675.283,E2 -9675.283} C_VEL
LIN {X 0,Y 425.248,Z 64.509,A -85,B 0,C 180,E1 -9678.618,E2 -9678.618} C_VEL
LIN {X 0,Y 425.27,Z 64.509,A -85,B 0,C 180,E1 -9682.304,E2 -9682.304} C_VEL
LIN {X 0,Y 425.285,Z 64.51,A -85,B 0,C 180,E1 -9685.815,E2 -9685.815} C_VEL
LIN {X 0,Y 425.287,Z 64.508,A -85,B 0,C 180,E1 -9689.24,E2 -9689.24} C_VEL
LIN {X 0,Y 425.24,Z 64.509,A -85,B 0,C 180,E1 -9692.434,E2 -9692.434} C_VEL
LIN {X 0,Y 425.321,Z 64.502,A -85,B 0,C 180,E1 -9695.6,E2 -9695.6} C_VEL
LIN {X 0,Y 425.296,Z 64.505,A -85,B 0,C 180,E1 -9698.681,E2 -9698.681} C_VEL
LIN {X 0,Y 425.323,Z 64.497,A -85,B 0,C 180,E1 -9701.702,E2 -9701.702} C_VEL
LIN {X 0,Y 425.338,Z 64.505,A -85,B 0,C 180,E1 -9704.67,E2 -9704.67} C_VEL
LIN {X 0,Y 425.415,Z 64.483,A -85,B 0,C 180,E1 -9707.598,E2 -9707.598} C_VEL
LIN {X 0,Y 425.409,Z 64.491,A -85,B 0,C 180,E1 -9711.449,E2 -9711.449} C_VEL
LIN {X 0,Y 425.508,Z 64.475,A -85,B 0,C 180,E1 -9714.312,E2 -9714.312} C_VEL
LIN {X 0,Y 425.571,Z 64.475,A -85,B 0,C 180,E1 -9718.107,E2 -9718.107} C_VEL
LIN {X 0,Y 425.512,Z 64.475,A -85,B 0,C 180,E1 -9720.946,E2 -9720.946} C_VEL
LIN {X 0,Y 425.517,Z 64.478,A -85,B 0,C 180,E1 -9722.84,E2 -9722.84} C_VEL
LIN {X 0,Y 425.53,Z 64.473,A -85,B 0,C 180,E1 -9725.687,E2 -9725.687} C_VEL
LIN {X 0,Y 425.409,Z 64.491,A -85,B 0,C 180,E1 -9728.551,E2 -9728.551} C_VEL
LIN {X 0,Y 425.415,Z 64.486,A -85,B 0,C 180,E1 -9732.402,E2 -9732.402} C_VEL
LIN {X 0,Y 425.388,Z 64.489,A -85,B 0,C 180,E1 -9736.312,E2 -9736.312} C_VEL
LIN {X 0,Y 425.331,Z 64.505,A -85,B 0,C 180,E1 -9739.635,E2 -9739.635} C_VEL
LIN {X 0,Y 425.306,Z 64.505,A -85,B 0,C 180,E1 -9743.365,E2 -9743.365} C_VEL
LIN {X 0,Y 425.343,Z 64.499,A -85,B 0,C 180,E1 -9746.842,E2 -9746.842} C_VEL
LIN {X 0,Y 425.293,Z 64.506,A -85,B 0,C 180,E1 -9749.719,E2 -9749.719} C_VEL
LIN {X 0,Y 425.285,Z 64.512,A -85,B 0,C 180,E1 -9753.048,E2 -9753.048} C_VEL
LIN {X 0,Y 425.285,Z 64.494,A -85,B 0,C 180,E1 -9755.928,E2 -9755.928} C_VEL
LIN {X 0,Y 425.29,Z 64.511,A -85,B 0,C 180,E1 -9759.042,E2 -9759.042} C_VEL
LIN {X 0,Y 425.292,Z 64.506,A -85,B 0,C 180,E1 -9761.958,E2 -9761.958} C_VEL
LIN {X 0,Y 425.287,Z 64.506,A -85,B 0,C 180,E1 -9765.283,E2 -9765.283} C_VEL
LIN {X 0,Y 425.278,Z 64.509,A -85,B 0,C 180,E1 -9768.621,E2 -9768.621} C_VEL
LIN {X 0,Y 425.315,Z 64.503,A -85,B 0,C 180,E1 -9771.103,E2 -9771.103} C_VEL
LIN {X 0,Y 425.302,Z 64.504,A -85,B 0,C 180,E1 -9774.664,E2 -9774.664} C_VEL
LIN {X 0,Y 425.268,Z 64.517,A -85,B 0,C 180,E1 -9778.073,E2 -9778.073} C_VEL
LIN {X 0,Y 425.383,Z 64.674,A -85,B 0,C 180,E1 -9781.573,E2 -9781.573} C_VEL
LIN {X 0,Y 427.975,Z 76.671,A -85,B 0,C 180,E1 -9784.157,E2 -9784.157} C_VEL
LIN {X 0,Y 428.753,Z 82.197,A -85,B 0,C 180,E1 -9785.292,E2 -9785.292} C_VEL
LIN {X 0,Y 427.517,Z 99.344,A -85,B 0,C 180,E1 -9788.545,E2 -9788.545} C_VEL
LIN {X 0,Y 426.816,Z 111.758,A -85,B 0,C 180,E1 -9790.876,E2 -9790.876} C_VEL
LIN {X 0,Y 430.837,Z 136.217,A -85,B 0,C 180,E1 -9791.524,E2 -9791.524} C_VEL
LIN {X 0,Y 431.148,Z 141.477,A -85,B 0,C 180,E1 -9791.631,E2 -9791.631} C_VEL
LIN {X 0,Y 430.262,Z 220.808,A -85,B 0,C 180,E1 -9792.993,E2 -9792.993} C_VEL
LIN {X 0,Y 429.615,Z 234.698,A -85,B 0,C 180,E1 -9793.425,E2 -9793.425} C_VEL
LIN {X 0,Y 428.968,Z 247.131,A -85,B 0,C 180,E1 -9794.011,E2 -9794.011} C_VEL
LIN {X 0,Y 428.172,Z 259.026,A -85,B 0,C 180,E1 -9794.774,E2 -9794.774} C_VEL
LIN {X 0,Y 427.354,Z 270.451,A -85,B 0,C 180,E1 -9795.718,E2 -9795.718} C_VEL
LIN {X 0,Y 426.552,Z 280.773,A -85,B 0,C 180,E1 -9796.785,E2 -9796.785} C_VEL
LIN {X 0,Y 425.967,Z 289.228,A -85,B 0,C 180,E1 -9797.856,E2 -9797.856} C_VEL
LIN {X 0,Y 425.202,Z 298.412,A -85,B 0,C 180,E1 -9799.283,E2 -9799.283} C_VEL
LIN {X 0,Y 424.73,Z 305.823,A -85,B 0,C 180,E1 -9800.715,E2 -9800.715} C_VEL
LIN {X 0,Y 424.37,Z 312.667,A -85,B 0,C 180,E1 -9802.386,E2 -9802.386} C_VEL
LIN {X 0,Y 424.235,Z 316.899,A -85,B 0,C 180,E1 -9803.71,E2 -9803.71} C_VEL
LIN {X 0,Y 424.192,Z 320.651,A -85,B 0,C 180,E1 -9805.248,E2 -9805.248} C_VEL
LIN {X 0,Y 424.177,Z 323.694,A -85,B 0,C 180,E1 -9807.151,E2 -9807.151} C_VEL
LIN {X 0,Y 424.167,Z 324.62,A -85,B 0,C 180,E1 -9808.101,E2 -9808.101} C_VEL
LIN {X 0,Y 424.142,Z 325.136,A -85,B 0,C 180,E1 -9809.05,E2 -9809.05} C_VEL
LIN {X 0,Y 424.145,Z 325.226,A -85,B 0,C 180,E1 -9810,E2 -9810} C_VEL
LIN {X 0,Y 424.168,Z 324.244,A -85,B 0,C 180,E1 -9811.899,E2 -9811.899} C_VEL
LIN {X 0,Y 424.217,Z 323.154,A -85,B 0,C 180,E1 -9812.849,E2 -9812.849} C_VEL
LIN {X 0,Y 424.13,Z 321.602,A -85,B 0,C 180,E1 -9813.8,E2 -9813.8} C_VEL
LIN {X 0,Y 424.203,Z 318.488,A -85,B 0,C 180,E1 -9815.228,E2 -9815.228} C_VEL
LIN {X 0,Y 424.223,Z 314.295,A -85,B 0,C 180,E1 -9816.659,E2 -9816.659} C_VEL
LIN {X 0,Y 424.488,Z 307.901,A -85,B 0,C 180,E1 -9818.329,E2 -9818.329} C_VEL
LIN {X 0,Y 424.805,Z 300.929,A -85,B 0,C 180,E1 -9819.763,E2 -9819.763} C_VEL
LIN {X 0,Y 425.172,Z 293.8,A -85,B 0,C 180,E1 -9820.958,E2 -9820.958} C_VEL
LIN {X 0,Y 425.711,Z 285.188,A -85,B 0,C 180,E1 -9822.151,E2 -9822.151} C_VEL
LIN {X 0,Y 426.339,Z 274.544,A -85,B 0,C 180,E1 -9823.343,E2 -9823.343} C_VEL
LIN {X 0,Y 426.948,Z 263.993,A -85,B 0,C 180,E1 -9824.295,E2 -9824.295} C_VEL
LIN {X 0,Y 427.654,Z 252.362,A -85,B 0,C 180,E1 -9825.122,E2 -9825.122} C_VEL
LIN {X 0,Y 428.269,Z 240.265,A -85,B 0,C 180,E1 -9825.771,E2 -9825.771} C_VEL
LIN {X 0,Y 428.794,Z 227.136,A -85,B 0,C 180,E1 -9826.27,E2 -9826.27} C_VEL
LIN {X 0,Y 429.058,Z 214.624,A -85,B 0,C 180,E1 -9826.566,E2 -9826.566} C_VEL
LIN {X 0,Y 429.7,Z 137.646,A -85,B 0,C 180,E1 -9827.849,E2 -9827.849} C_VEL
LIN {X 0,Y 426.204,Z 111.976,A -85,B 0,C 180,E1 -9828.445,E2 -9828.445} C_VEL
LIN {X 0,Y 427.181,Z 92.733,A -85,B 0,C 180,E1 -9831.98,E2 -9831.98} C_VEL
LIN {X 0,Y 427.984,Z 79.158,A -85,B 0,C 180,E1 -9834.496,E2 -9834.496} C_VEL
LIN {X 0,Y 426.646,Z 70.844,A -85,B 0,C 180,E1 -9836.145,E2 -9836.145} C_VEL
LIN {X 0,Y 425.401,Z 64.492,A -85,B 0,C 180,E1 -9837.467,E2 -9837.467} C_VEL
LIN {X 0,Y 425.288,Z 64.506,A -85,B 0,C 180,E1 -9840.816,E2 -9840.816} C_VEL
LIN {X 0,Y 425.311,Z 64.505,A -85,B 0,C 180,E1 -9844.288,E2 -9844.288} C_VEL
LIN {X 0,Y 425.286,Z 64.512,A -85,B 0,C 180,E1 -9847.693,E2 -9847.693} C_VEL
LIN {X 0,Y 425.284,Z 64.506,A -85,B 0,C 180,E1 -9850.521,E2 -9850.521} C_VEL
LIN {X 0,Y 425.257,Z 64.514,A -85,B 0,C 180,E1 -9853.351,E2 -9853.351} C_VEL
LIN {X 0,Y 425.256,Z 64.509,A -85,B 0,C 180,E1 -9856.649,E2 -9856.649} C_VEL
LIN {X 0,Y 425.285,Z 64.507,A -85,B 0,C 180,E1 -9859.873,E2 -9859.873} C_VEL
LIN {X 0,Y 425.277,Z 64.507,A -85,B 0,C 180,E1 -9862.488,E2 -9862.488} C_VEL
LIN {X 0,Y 425.307,Z 64.504,A -85,B 0,C 180,E1 -9865.817,E2 -9865.817} C_VEL
LIN {X 0,Y 425.29,Z 64.51,A -85,B 0,C 180,E1 -9869.239,E2 -9869.239} C_VEL
LIN {X 0,Y 425.348,Z 64.5,A -85,B 0,C 180,E1 -9872.442,E2 -9872.442} C_VEL
LIN {X 0,Y 425.35,Z 64.498,A -85,B 0,C 180,E1 -9875.602,E2 -9875.602} C_VEL
LIN {X 0,Y 425.293,Z 64.511,A -85,B 0,C 180,E1 -9878.682,E2 -9878.682} C_VEL
LIN {X 0,Y 425.321,Z 64.501,A -85,B 0,C 180,E1 -9881.702,E2 -9881.702} C_VEL
LIN {X 0,Y 425.348,Z 64.504,A -85,B 0,C 180,E1 -9884.671,E2 -9884.671} C_VEL
LIN {X 0,Y 425.411,Z 64.49,A -85,B 0,C 180,E1 -9887.598,E2 -9887.598} C_VEL
LIN {X 0,Y 425.442,Z 64.486,A -85,B 0,C 180,E1 -9891.45,E2 -9891.45} C_VEL
LIN {X 0,Y 425.55,Z 64.48,A -85,B 0,C 180,E1 -9894.313,E2 -9894.313} C_VEL
LIN {X 0,Y 425.57,Z 64.477,A -85,B 0,C 180,E1 -9898.107,E2 -9898.107} C_VEL
LIN {X 0,Y 425.699,Z 64.46,A -85,B 0,C 180,E1 -9900,E2 -9900} C_VEL
LIN {X 0,Y 425.538,Z 64.474,A -85,B 0,C 180,E1 -9902.84,E2 -9902.84} C_VEL
LIN {X 0,Y 425.497,Z 64.479,A -85,B 0,C 180,E1 -9906.517,E2 -9906.517} C_VEL
LIN {X 0,Y 425.398,Z 64.495,A -85,B 0,C 180,E1 -9909.51,E2 -9909.51} C_VEL
LIN {X 0,Y 425.393,Z 64.492,A -85,B 0,C 180,E1 -9912.904,E2 -9912.904} C_VEL
LIN {X 0,Y 425.361,Z 64.496,A -85,B 0,C 180,E1 -9916.605,E2 -9916.605} C_VEL
LIN {X 0,Y 425.328,Z 64.506,A -85,B 0,C 180,E1 -9919.636,E2 -9919.636} C_VEL
LIN {X 0,Y 425.304,Z 64.511,A -85,B 0,C 180,E1 -9923.366,E2 -9923.366} C_VEL
LIN {X 0,Y 425.34,Z 64.501,A -85,B 0,C 180,E1 -9926.843,E2 -9926.843} C_VEL
LIN {X 0,Y 425.291,Z 64.506,A -85,B 0,C 180,E1 -9929.72,E2 -9929.72} C_VEL
LIN {X 0,Y 425.282,Z 64.513,A -85,B 0,C 180,E1 -9933.048,E2 -9933.048} C_VEL
LIN {X 0,Y 425.282,Z 64.506,A -85,B 0,C 180,E1 -9935.929,E2 -9935.929} C_VEL
LIN {X 0,Y 425.266,Z 64.513,A -85,B 0,C 180,E1 -9939.038,E2 -9939.038} C_VEL
LIN {X 0,Y 425.261,Z 64.515,A -85,B 0,C 180,E1 -9942.655,E2 -9942.655} C_VEL
LIN {X 0,Y 425.286,Z 64.507,A -85,B 0,C 180,E1 -9945.284,E2 -9945.284} C_VEL
LIN {X 0,Y 425.267,Z 64.515,A -85,B 0,C 180,E1 -9948.621,E2 -9948.621} C_VEL
LIN {X 0,Y 425.282,Z 64.507,A -85,B 0,C 180,E1 -9951.1,E2 -9951.1} C_VEL
LIN {X 0,Y 425.3,Z 64.507,A -85,B 0,C 180,E1 -9954.664,E2 -9954.664} C_VEL
LIN {X 0,Y 425.268,Z 64.513,A -85,B 0,C 180,E1 -9958.074,E2 -9958.074} C_VEL
LIN {X 0,Y 425.316,Z 64.502,A -85,B 0,C 180,E1 -9961.367,E2 -9961.367} C_VEL
LIN {X 0,Y 425.265,Z 64.51,A -85,B 0,C 180,E1 -9964.553,E2 -9964.553} C_VEL
LIN {X 0,Y 425.282,Z 64.507,A -85,B 0,C 180,E1 -9966.634,E2 -9966.634} C_VEL
LIN {X 0,Y 425.299,Z 64.509,A -85,B 0,C 180,E1 -9969.695,E2 -9969.695} C_VEL
LIN {X 0,Y 425.342,Z 64.501,A -85,B 0,C 180,E1 -9972.698,E2 -9972.698} C_VEL
LIN {X 0,Y 425.381,Z 64.538,A -85,B 0,C 180,E1 -9975.835,E2 -9975.835} C_VEL
LIN {X 0,Y 426.737,Z 73.036,A -85,B 0,C 180,E1 -9977.879,E2 -9977.879} C_VEL
LIN {X 0,Y 426.801,Z 76.711,A -85,B 0,C 180,E1 -9978.691,E2 -9978.691} C_VEL
LIN {X 0,Y 430.167,Z 94.26,A -85,B 0,C 180,E1 -9979.123,E2 -9979.123} C_VEL
LIN {X 0,Y 429.151,Z 183.732,A -85,B 0,C 180,E1 -9980.634,E2 -9980.634} C_VEL
LIN {X 0,Y 428.918,Z 196.714,A -85,B 0,C 180,E1 -9981.045,E2 -9981.045} C_VEL
LIN {X 0,Y 428.764,Z 200.225,A -85,B 0,C 180,E1 -9981.186,E2 -9981.186} C_VEL
LIN {X 0,Y 427.869,Z 205.892,A -85,B 0,C 180,E1 -9981.428,E2 -9981.428} C_VEL
LIN {X 0,Y 423.466,Z 218.303,A -85,B 0,C 180,E1 -9982.027,E2 -9982.027} C_VEL
LIN {X 0,Y 421.273,Z 225.126,A -85,B 0,C 180,E1 -9982.468,E2 -9982.468} C_VEL
LIN {X 0,Y 420.759,Z 228.414,A -85,B 0,C 180,E1 -9982.732,E2 -9982.732} C_VEL
LIN {X 0,Y 420.111,Z 239.158,A -85,B 0,C 180,E1 -9983.758,E2 -9983.758} C_VEL
LIN {X 0,Y 419.415,Z 249.162,A -85,B 0,C 180,E1 -9984.953,E2 -9984.953} C_VEL
LIN {X 0,Y 418.771,Z 258.809,A -85,B 0,C 180,E1 -9986.392,E2 -9986.392} C_VEL
LIN {X 0,Y 418.166,Z 266.556,A -85,B 0,C 180,E1 -9987.833,E2 -9987.833} C_VEL
LIN {X 0,Y 417.739,Z 273.638,A -85,B 0,C 180,E1 -9989.518,E2 -9989.518} C_VEL
LIN {X 0,Y 417.39,Z 278.385,A -85,B 0,C 180,E1 -9990.965,E2 -9990.965} C_VEL
LIN {X 0,Y 417.304,Z 282.021,A -85,B 0,C 180,E1 -9992.413,E2 -9992.413} C_VEL
LIN {X 0,Y 417.146,Z 284.666,A -85,B 0,C 180,E1 -9993.864,E2 -9993.864} C_VEL
LIN {X 0,Y 417.132,Z 285.913,A -85,B 0,C 180,E1 -9994.833,E2 -9994.833} C_VEL
LIN {X 0,Y 417.197,Z 287.024,A -85,B 0,C 180,E1 -9996.327,E2 -9996.327} C_VEL
LIN {X 0,Y 417.093,Z 287.217,A -85,B 0,C 180,E1 -9997.747,E2 -9997.747} C_VEL
LIN {X 0,Y 417.09,Z 286.87,A -85,B 0,C 180,E1 -9998.723,E2 -9998.723} C_VEL
LIN {X 0,Y 417.094,Z 286.128,A -85,B 0,C 180,E1 -9999.701,E2 -9999.701} C_VEL
LIN {X 0,Y 417.19,Z 284.937,A -85,B 0,C 180,E1 -10000.679,E2 -10000.679} C_VEL
LIN {X 0,Y 417.501,Z 281.658,A -85,B 0,C 180,E1 -10002.485,E2 -10002.485} C_VEL
LIN {X 0,Y 417.807,Z 277.38,A -85,B 0,C 180,E1 -10004.118,E2 -10004.118} C_VEL
LIN {X 0,Y 418.353,Z 271.257,A -85,B 0,C 180,E1 -10005.842,E2 -10005.842} C_VEL
LIN {X 0,Y 418.905,Z 264.296,A -85,B 0,C 180,E1 -10007.372,E2 -10007.372} C_VEL
LIN {X 0,Y 419.636,Z 256.121,A -85,B 0,C 180,E1 -10008.808,E2 -10008.808} C_VEL
LIN {X 0,Y 420.376,Z 247.402,A -85,B 0,C 180,E1 -10010.043,E2 -10010.043} C_VEL
LIN {X 0,Y 421.154,Z 236.602,A -85,B 0,C 180,E1 -10011.282,E2 -10011.282} C_VEL
LIN {X 0,Y 421.966,Z 225.798,A -85,B 0,C 180,E1 -10012.267,E2 -10012.267} C_VEL
LIN {X 0,Y 422.735,Z 213.606,A -85,B 0,C 180,E1 -10013.127,E2 -10013.127} C_VEL
LIN {X 0,Y 423.367,Z 201.024,A -85,B 0,C 180,E1 -10013.792,E2 -10013.792} C_VEL
LIN {X 0,Y 423.793,Z 188.836,A -85,B 0,C 180,E1 -10014.244,E2 -10014.244} C_VEL
LIN {X 0,Y 424.074,Z 173.529,A -85,B 0,C 180,E1 -10014.574,E2 -10014.574} C_VEL
LIN {X 0,Y 425.007,Z 95.632,A -85,B 0,C 180,E1 -10015.909,E2 -10015.909} C_VEL
LIN {X 0,Y 420.472,Z 77.282,A -85,B 0,C 180,E1 -10016.484,E2 -10016.484} C_VEL
LIN {X 0,Y 419.034,Z 69.015,A -85,B 0,C 180,E1 -10018.555,E2 -10018.555} C_VEL
LIN {X 0,Y 418.261,Z 65.387,A -85,B 0,C 180,E1 -10019.507,E2 -10019.507} C_VEL
LIN {X 0,Y 418.245,Z 65.388,A -85,B 0,C 180,E1 -10022.84,E2 -10022.84} C_VEL
LIN {X 0,Y 418.241,Z 65.39,A -85,B 0,C 180,E1 -10026.236,E2 -10026.236} C_VEL
LIN {X 0,Y 418.2,Z 65.394,A -85,B 0,C 180,E1 -10029.688,E2 -10029.688} C_VEL
LIN {X 0,Y 418.209,Z 65.392,A -85,B 0,C 180,E1 -10032.317,E2 -10032.317} C_VEL
LIN {X 0,Y 418.237,Z 65.375,A -85,B 0,C 180,E1 -10035.108,E2 -10035.108} C_VEL
LIN {X 0,Y 418.22,Z 65.39,A -85,B 0,C 180,E1 -10037.764,E2 -10037.764} C_VEL
LIN {X 0,Y 418.229,Z 65.388,A -85,B 0,C 180,E1 -10041.555,E2 -10041.555} C_VEL
LIN {X 0,Y 418.25,Z 65.383,A -85,B 0,C 180,E1 -10045.158,E2 -10045.158} C_VEL
LIN {X 0,Y 418.234,Z 65.386,A -85,B 0,C 180,E1 -10047.47,E2 -10047.47} C_VEL
LIN {X 0,Y 418.26,Z 65.385,A -85,B 0,C 180,E1 -10050.898,E2 -10050.898} C_VEL
LIN {X 0,Y 418.213,Z 65.387,A -85,B 0,C 180,E1 -10054.092,E2 -10054.092} C_VEL
LIN {X 0,Y 418.23,Z 65.383,A -85,B 0,C 180,E1 -10057.263,E2 -10057.263} C_VEL
LIN {X 0,Y 418.287,Z 65.38,A -85,B 0,C 180,E1 -10060.364,E2 -10060.364} C_VEL
LIN {X 0,Y 418.319,Z 65.373,A -85,B 0,C 180,E1 -10063.404,E2 -10063.404} C_VEL
LIN {X 0,Y 418.35,Z 65.366,A -85,B 0,C 180,E1 -10066.999,E2 -10066.999} C_VEL
LIN {X 0,Y 418.337,Z 65.375,A -85,B 0,C 180,E1 -10070.328,E2 -10070.328} C_VEL
LIN {X 0,Y 418.439,Z 65.352,A -85,B 0,C 180,E1 -10073.248,E2 -10073.248} C_VEL
LIN {X 0,Y 418.321,Z 65.372,A -85,B 0,C 180,E1 -10075.181,E2 -10075.181} C_VEL
LIN {X 0,Y 418.54,Z 65.351,A -85,B 0,C 180,E1 -10078.075,E2 -10078.075} C_VEL
LIN {X 0,Y 418.475,Z 65.352,A -85,B 0,C 180,E1 -10080.962,E2 -10080.962} C_VEL
LIN {X 0,Y 418.474,Z 65.355,A -85,B 0,C 180,E1 -10082.888,E2 -10082.888} C_VEL
LIN {X 0,Y 418.487,Z 65.349,A -85,B 0,C 180,E1 -10085.783,E2 -10085.783} C_VEL
LIN {X 0,Y 418.379,Z 65.366,A -85,B 0,C 180,E1 -10088.695,E2 -10088.695} C_VEL
LIN {X 0,Y 418.317,Z 65.371,A -85,B 0,C 180,E1 -10091.631,E2 -10091.631} C_VEL
LIN {X 0,Y 418.301,Z 65.376,A -85,B 0,C 180,E1 -10094.597,E2 -10094.597} C_VEL
LIN {X 0,Y 418.28,Z 65.377,A -85,B 0,C 180,E1 -10097.604,E2 -10097.604} C_VEL
LIN {X 0,Y 418.252,Z 65.382,A -85,B 0,C 180,E1 -10100.663,E2 -10100.663} C_VEL
LIN {X 0,Y 418.287,Z 65.381,A -85,B 0,C 180,E1 -10103.781,E2 -10103.781} C_VEL
LIN {X 0,Y 418.313,Z 65.374,A -85,B 0,C 180,E1 -10107.07,E2 -10107.07} C_VEL
LIN {X 0,Y 418.247,Z 65.382,A -85,B 0,C 180,E1 -10110.272,E2 -10110.272} C_VEL
LIN {X 0,Y 418.251,Z 65.382,A -85,B 0,C 180,E1 -10113.677,E2 -10113.677} C_VEL
LIN {X 0,Y 418.242,Z 65.375,A -85,B 0,C 180,E1 -10117.224,E2 -10117.224} C_VEL
LIN {X 0,Y 418.249,Z 65.384,A -85,B 0,C 180,E1 -10119.682,E2 -10119.682} C_VEL
LIN {X 0,Y 418.232,Z 65.388,A -85,B 0,C 180,E1 -10122.321,E2 -10122.321} C_VEL
LIN {X 0,Y 418.238,Z 65.385,A -85,B 0,C 180,E1 -10125.108,E2 -10125.108} C_VEL
LIN {X 0,Y 418.243,Z 65.384,A -85,B 0,C 180,E1 -10127.767,E2 -10127.767} C_VEL
LIN {X 0,Y 418.261,Z 65.384,A -85,B 0,C 180,E1 -10130.618,E2 -10130.618} C_VEL
LIN {X 0,Y 418.246,Z 65.385,A -85,B 0,C 180,E1 -10133.976,E2 -10133.976} C_VEL
LIN {X 0,Y 418.26,Z 65.388,A -85,B 0,C 180,E1 -10137.156,E2 -10137.156} C_VEL
LIN {X 0,Y 418.271,Z 65.387,A -85,B 0,C 180,E1 -10140.895,E2 -10140.895} C_VEL
LIN {X 0,Y 418.311,Z 65.514,A -85,B 0,C 180,E1 -10141.237,E2 -10141.237} C_VEL
LIN {X 0,Y 420.806,Z 76.823,A -85,B 0,C 180,E1 -10143.731,E2 -10143.731} C_VEL
LIN {X 0,Y 421.875,Z 83.429,A -85,B 0,C 180,E1 -10145.125,E2 -10145.125} C_VEL
LIN {X 0,Y 420.667,Z 99.242,A -85,B 0,C 180,E1 -10148.178,E2 -10148.178} C_VEL
LIN {X 0,Y 419.913,Z 111.464,A -85,B 0,C 180,E1 -10150.514,E2 -10150.514} C_VEL
LIN {X 0,Y 424.041,Z 135.936,A -85,B 0,C 180,E1 -10151.178,E2 -10151.178} C_VEL
LIN {X 0,Y 424.52,Z 140.915,A -85,B 0,C 180,E1 -10151.291,E2 -10151.291} C_VEL
LIN {X 0,Y 423.563,Z 220.745,A -85,B 0,C 180,E1 -10152.684,E2 -10152.684} C_VEL
LIN {X 0,Y 422.896,Z 234.547,A -85,B 0,C 180,E1 -10153.123,E2 -10153.123} C_VEL
LIN {X 0,Y 422.172,Z 247.437,A -85,B 0,C 180,E1 -10153.747,E2 -10153.747} C_VEL
LIN {X 0,Y 421.337,Z 259.184,A -85,B 0,C 180,E1 -10154.521,E2 -10154.521} C_VEL
LIN {X 0,Y 420.473,Z 270.521,A -85,B 0,C 180,E1 -10155.48,E2 -10155.48} C_VEL
LIN {X 0,Y 419.615,Z 280.765,A -85,B 0,C 180,E1 -10156.562,E2 -10156.562} C_VEL
LIN {X 0,Y 419.007,Z 289.163,A -85,B 0,C 180,E1 -10157.651,E2 -10157.651} C_VEL
LIN {X 0,Y 418.208,Z 298.29,A -85,B 0,C 180,E1 -10159.102,E2 -10159.102} C_VEL
LIN {X 0,Y 417.701,Z 305.664,A -85,B 0,C 180,E1 -10160.558,E2 -10160.558} C_VEL
LIN {X 0,Y 417.317,Z 312.462,A -85,B 0,C 180,E1 -10162.257,E2 -10162.257} C_VEL
LIN {X 0,Y 417.158,Z 316.977,A -85,B 0,C 180,E1 -10163.718,E2 -10163.718} C_VEL
LIN {X 0,Y 417.096,Z 320.394,A -85,B 0,C 180,E1 -10165.167,E2 -10165.167} C_VEL
LIN {X 0,Y 417.073,Z 323.413,A -85,B 0,C 180,E1 -10167.102,E2 -10167.102} C_VEL
LIN {X 0,Y 417.093,Z 324.328,A -85,B 0,C 180,E1 -10168.068,E2 -10168.068} C_VEL
LIN {X 0,Y 417.062,Z 324.822,A -85,B 0,C 180,E1 -10169.034,E2 -10169.034} C_VEL
LIN {X 0,Y 417.061,Z 324.9,A -85,B 0,C 180,E1 -10170,E2 -10170} C_VEL
LIN {X 0,Y 417.095,Z 323.896,A -85,B 0,C 180,E1 -10171.931,E2 -10171.931} C_VEL
LIN {X 0,Y 417.114,Z 322.783,A -85,B 0,C 180,E1 -10172.897,E2 -10172.897} C_VEL
LIN {X 0,Y 417.042,Z 321.217,A -85,B 0,C 180,E1 -10173.865,E2 -10173.865} C_VEL
LIN {X 0,Y 417.111,Z 318.077,A -85,B 0,C 180,E1 -10175.317,E2 -10175.317} C_VEL
LIN {X 0,Y 417.158,Z 313.858,A -85,B 0,C 180,E1 -10176.772,E2 -10176.772} C_VEL
